  MoveL 1350 to (235.6, 160.89, 31.63) mm, rotated rx 180 ry 0 rz 180 deg; joints [-30.149, 31.04, 26.19, 47.019, 43.356, -37.963]
  Call Extruder(260.06527)
  MoveL 1351 to (235.35, 161.1, 31.63) mm, rotated rx -180 ry 0 rz 180 deg; joints [-30.182, 30.989, 26.274, 47.082, 43.354, -38.025]
  Call Extruder(260.39930)
  MoveL 1352 to (234.9, 161.43, 31.63) mm, rotated rx 180 ry 0 rz 180 deg; joints [-30.234, 30.885, 26.445, 47.194, 43.341, -38.14]
  MoveL 1353 to (234.9, 161.43, 31.63) mm, rotated rx 180 ry 0 rz 180 deg; joints [-30.234, 30.885, 26.445, 47.194, 43.341, -38.14]
  Call Extruder(260.73214)
  MoveL 1354 to (234.45, 161.76, 31.63) mm, rotated rx 180 ry 0 rz 180 deg; joints [-30.287, 30.782, 26.613, 47.306, 43.329, -38.255]
  MoveL 1355 to (234.45, 161.76, 31.63) mm, rotated rx 180 ry 0 rz 180 deg; joints [-30.287, 30.782, 26.613, 47.306, 43.329, -38.255]
  Call Extruder(260.91134)
  MoveL 1356 to (234.21, 161.94, 31.63) mm, rotated rx 180 ry 0 rz 180 deg; joints [-30.316, 30.726, 26.705, 47.366, 43.322, -38.316]
  MoveL 1357 to (234.21, 161.94, 31.63) mm, rotated rx 180 ry 0 rz 180 deg; joints [-30.316, 30.726, 26.705, 47.366, 43.322, -38.316]
  Call Extruder(261.11946)
  MoveL 1358 to (233.9, 162.11, 31.63) mm, rotated rx 180 ry 0 rz 180 deg; joints [-30.347, 30.648, 26.833, 47.441, 43.308, -38.396]
  MoveL 1359 to (233.9, 162.11, 31.63) mm, rotated rx 180 ry 0 rz 180 deg; joints [-30.347, 30.648, 26.833, 47.441, 43.308, -38.396]
  Call Extruder(261.32679)
  MoveL 1360 to (233.6, 162.29, 31.63) mm, rotated rx -180 ry 0 rz -180 deg; joints [-30.379, 30.57, 26.96, 47.515, 43.295, -38.475]
  MoveL 1361 to (233.6, 162.29, 31.63) mm, rotated rx -180 ry 0 rz -180 deg; joints [-30.379, 30.57, 26.96, 47.515, 43.295, -38.475]
  Call Extruder(261.53335)
  MoveL 1362 to (233.29, 162.46, 31.63) mm, rotated rx -180 ry 0 rz 180 deg; joints [-30.41, 30.494, 27.085, 47.589, 43.281, -38.554]
  MoveL 1363 to (233.29, 162.46, 31.63) mm, rotated rx -180 ry 0 rz 180 deg; joints [-30.41, 30.494, 27.085, 47.589, 43.281, -38.554]
  Call Extruder(261.73913)
  MoveL 1364 to (232.99, 162.64, 31.63) mm, rotated rx -180 ry 0 rz 180 deg; joints [-30.442, 30.417, 27.21, 47.663, 43.269, -38.632]
  MoveL 1365 to (232.99, 162.64, 31.63) mm, rotated rx -180 ry 0 rz 180 deg; joints [-30.442, 30.417, 27.21, 47.663, 43.269, -38.632]
  Call Extruder(261.89741)
  MoveL 1366 to (232.74, 162.74, 31.63) mm, rotated rx 180 ry 0 rz -180 deg; joints [-30.464, 30.347, 27.324, 47.724, 43.253, -38.698]
  MoveL 1367 to (232.74, 162.74, 31.63) mm, rotated rx 180 ry 0 rz -180 deg; joints [-30.464, 30.347, 27.324, 47.724, 43.253, -38.698]
  Call Extruder(262.05508)
  MoveL 1368 to (232.49, 162.85, 31.63) mm, rotated rx -180 ry 0 rz 180 deg; joints [-30.487, 30.277, 27.438, 47.784, 43.238, -38.764]
  MoveL 1369 to (232.49, 162.85, 31.63) mm, rotated rx -180 ry 0 rz 180 deg; joints [-30.487, 30.277, 27.438, 47.784, 43.238, -38.764]
  Call Extruder(262.22517)
  MoveL 1370 to (232.22, 162.97, 31.63) mm, rotated rx 180 ry 0 rz -180 deg; joints [-30.511, 30.202, 27.56, 47.849, 43.222, -38.835]
  MoveL 1371 to (232.22, 162.97, 31.63) mm, rotated rx 180 ry 0 rz -180 deg; joints [-30.511, 30.202, 27.56, 47.849, 43.222, -38.835]
  Call Extruder(262.40753)
  MoveL 1372 to (231.93, 163.09, 31.63) mm, rotated rx 180 ry 0 rz 180 deg; joints [-30.538, 30.12, 27.692, 47.918, 43.204, -38.912]
  MoveL 1373 to (231.93, 163.09, 31.63) mm, rotated rx 180 ry 0 rz 180 deg; joints [-30.538, 30.12, 27.692, 47.918, 43.204, -38.912]
  Call Extruder(262.58914)
  MoveL 1374 to (231.64, 163.21, 31.63) mm, rotated rx 180 ry 0 rz 180 deg; joints [-30.564, 30.04, 27.823, 47.988, 43.187, -38.988]
  MoveL 1375 to (231.64, 163.21, 31.63) mm, rotated rx 180 ry 0 rz 180 deg; joints [-30.564, 30.04, 27.823, 47.988, 43.187, -38.988]
  Call Extruder(262.70258)
  MoveL 1376 to (231.45, 163.27, 31.63) mm, rotated rx -180 ry 0 rz 180 deg; joints [-30.579, 29.984, 27.912, 48.032, 43.174, -39.038]
  MoveL 1377 to (231.45, 163.27, 31.63) mm, rotated rx -180 ry 0 rz 180 deg; joints [-30.579, 29.984, 27.912, 48.032, 43.174, -39.038]
  Call Extruder(262.81558)
  MoveL 1378 to (231.26, 163.33, 31.63) mm, rotated rx 180 ry 0 rz 180 deg; joints [-30.595, 29.929, 28.002, 48.077, 43.161, -39.087]
  MoveL 1379 to (231.26, 163.33, 31.63) mm, rotated rx 180 ry 0 rz 180 deg; joints [-30.595, 29.929, 28.002, 48.077, 43.161, -39.087]
  Call Extruder(262.92814)
  MoveL 1380 to (231.07, 163.39, 31.63) mm, rotated rx 180 ry 0 rz 180 deg; joints [-30.61, 29.875, 28.09, 48.121, 43.148, -39.137]
  MoveL 1381 to (231.07, 163.39, 31.63) mm, rotated rx 180 ry 0 rz 180 deg; joints [-30.61, 29.875, 28.09, 48.121, 43.148, -39.137]
  Call Extruder(263.04025)
  MoveL 1382 to (230.88, 163.45, 31.63) mm, rotated rx 180 ry 0 rz 180 deg; joints [-30.625, 29.82, 28.178, 48.165, 43.135, -39.186]
  MoveL 1383 to (230.88, 163.45, 31.63) mm, rotated rx 180 ry 0 rz 180 deg; joints [-30.625, 29.82, 28.178, 48.165, 43.135, -39.186]
  Call Extruder(263.15191)
  MoveL 1384 to (230.7, 163.51, 31.63) mm, rotated rx 180 ry 0 rz 180 deg; joints [-30.641, 29.766, 28.265, 48.209, 43.123, -39.235]
  MoveL 1385 to (230.7, 163.51, 31.63) mm, rotated rx 180 ry 0 rz 180 deg; joints [-30.641, 29.766, 28.265, 48.209, 43.123, -39.235]
  Call Extruder(263.28301)
  MoveL 1386 to (230.47, 163.58, 31.63) mm, rotated rx 180 ry 0 rz 180 deg; joints [-30.659, 29.701, 28.37, 48.261, 43.108, -39.293]
  MoveL 1387 to (230.47, 163.58, 31.63) mm, rotated rx 180 ry 0 rz 180 deg; joints [-30.659, 29.701, 28.37, 48.261, 43.108, -39.293]
  Call Extruder(263.41354)
  MoveL 1388 to (230.25, 163.65, 31.63) mm, rotated rx 180 ry 0 rz -180 deg; joints [-30.677, 29.636, 28.474, 48.313, 43.093, -39.351]
  MoveL 1389 to (230.25, 163.65, 31.63) mm, rotated rx 180 ry 0 rz -180 deg; joints [-30.677, 29.636, 28.474, 48.313, 43.093, -39.351]
  Call Extruder(263.54350)
  MoveL 1390 to (230.02, 163.72, 31.63) mm, rotated rx -180 ry 0 rz 180 deg; joints [-30.694, 29.572, 28.577, 48.364, 43.078, -39.408]
  MoveL 1391 to (230.02, 163.72, 31.63) mm, rotated rx -180 ry 0 rz 180 deg; joints [-30.694, 29.572, 28.577, 48.364, 43.078, -39.408]
  Call Extruder(263.67290)
  MoveL 1392 to (229.8, 163.78, 31.63) mm, rotated rx 180 ry 0 rz 180 deg; joints [-30.712, 29.508, 28.68, 48.415, 43.064, -39.466]
  MoveL 1393 to (229.8, 163.78, 31.63) mm, rotated rx 180 ry 0 rz 180 deg; joints [-30.712, 29.508, 28.68, 48.415, 43.064, -39.466]
  Call Extruder(263.79488)
  MoveL 1394 to (229.59, 163.84, 31.63) mm, rotated rx 180 ry 0 rz 180 deg; joints [-30.729, 29.445, 28.78, 48.464, 43.049, -39.521]
  MoveL 1395 to (229.59, 163.84, 31.63) mm, rotated rx 180 ry 0 rz 180 deg; joints [-30.729, 29.445, 28.78, 48.464, 43.049, -39.521]
  Call Extruder(263.90973)
  MoveL 1396 to (229.38, 163.88, 31.63) mm, rotated rx 180 ry 0 rz 180 deg; joints [-30.744, 29.384, 28.878, 48.511, 43.034, -39.573]
  MoveL 1397 to (229.38, 163.88, 31.63) mm, rotated rx 180 ry 0 rz 180 deg; joints [-30.744, 29.384, 28.878, 48.511, 43.034, -39.573]
  Call Extruder(264.02412)
  MoveL 1398 to (229.18, 163.93, 31.63) mm, rotated rx 180 ry 0 rz 180 deg; joints [-30.758, 29.324, 28.976, 48.557, 43.019, -39.626]
  MoveL 1399 to (229.18, 163.93, 31.63) mm, rotated rx 180 ry 0 rz 180 deg; joints [-30.758, 29.324, 28.976, 48.557, 43.019, -39.626]
  Call Extruder(264.13806)
  MoveL 1400 to (228.97, 163.97, 31.63) mm, rotated rx -180 ry 0 rz 180 deg; joints [-30.773, 29.263, 29.073, 48.603, 43.005, -39.678]
  MoveL 1401 to (228.97, 163.97, 31.63) mm, rotated rx -180 ry 0 rz 180 deg; joints [-30.773, 29.263, 29.073, 48.603, 43.005, -39.678]
  Call Extruder(264.25155)
  MoveL 1402 to (228.77, 164.02, 31.63) mm, rotated rx 180 ry 0 rz 180 deg; joints [-30.788, 29.203, 29.169, 48.648, 42.99, -39.73]
  MoveL 1403 to (228.77, 164.02, 31.63) mm, rotated rx 180 ry 0 rz 180 deg; joints [-30.788, 29.203, 29.169, 48.648, 42.99, -39.73]
  Call Extruder(264.38884)
  MoveL 1404 to (228.52, 164.07, 31.63) mm, rotated rx 180 ry 0 rz 180 deg; joints [-30.806, 29.129, 29.287, 48.704, 42.973, -39.793]
  MoveL 1405 to (228.52, 164.07, 31.63) mm, rotated rx 180 ry 0 rz 180 deg; joints [-30.806, 29.129, 29.287, 48.704, 42.973, -39.793]
  Call Extruder(264.52551)
  MoveL 1406 to (228.27, 164.12, 31.63) mm, rotated rx -180 ry 0 rz 180 deg; joints [-30.823, 29.055, 29.404, 48.759, 42.955, -39.856]
  MoveL 1407 to (228.27, 164.12, 31.63) mm, rotated rx -180 ry 0 rz 180 deg; joints [-30.823, 29.055, 29.404, 48.759, 42.955, -39.856]
  Call Extruder(264.66157)
  MoveL 1408 to (228.02, 164.17, 31.63) mm, rotated rx -180 ry 0 rz 180 deg; joints [-30.841, 28.982, 29.52, 48.814, 42.938, -39.919]
  MoveL 1409 to (228.02, 164.17, 31.63) mm, rotated rx -180 ry 0 rz 180 deg; joints [-30.841, 28.982, 29.52, 48.814, 42.938, -39.919]
  Call Extruder(264.79703)
  MoveL 1410 to (227.77, 164.22, 31.63) mm, rotated rx -180 ry 0 rz -180 deg; joints [-30.859, 28.91, 29.636, 48.869, 42.921, -39.981]
  MoveL 1411 to (227.77, 164.22, 31.63) mm, rotated rx -180 ry 0 rz -180 deg; joints [-30.859, 28.91, 29.636, 48.869, 42.921, -39.981]
  Call Extruder(264.93187)
  MoveL 1412 to (227.52, 164.27, 31.63) mm, rotated rx 180 ry 0 rz 180 deg; joints [-30.877, 28.838, 29.751, 48.923, 42.905, -40.042]
  MoveL 1413 to (227.52, 164.27, 31.63) mm, rotated rx 180 ry 0 rz 180 deg; joints [-30.877, 28.838, 29.751, 48.923, 42.905, -40.042]
  Call Extruder(265.06610)
  MoveL 1414 to (227.27, 164.32, 31.63) mm, rotated rx 180 ry 0 rz 180 deg; joints [-30.895, 28.766, 29.864, 48.978, 42.888, -40.104]
  MoveL 1415 to (227.27, 164.32, 31.63) mm, rotated rx 180 ry 0 rz 180 deg; joints [-30.895, 28.766, 29.864, 48.978, 42.888, -40.104]
  Call Extruder(265.19972)
  MoveL 1416 to (227.02, 164.36, 31.63) mm, rotated rx -180 ry 0 rz -180 deg; joints [-30.912, 28.695, 29.978, 49.032, 42.872, -40.165]
  MoveL 1417 to (227.02, 164.36, 31.63) mm, rotated rx -180 ry 0 rz -180 deg; joints [-30.912, 28.695, 29.978, 49.032, 42.872, -40.165]
  Call Extruder(265.36183)
  MoveL 1418 to (226.72, 164.41, 31.63) mm, rotated rx -180 ry 0 rz 180 deg; joints [-30.933, 28.606, 30.119, 49.097, 42.851, -40.24]
  MoveL 1419 to (226.72, 164.41, 31.63) mm, rotated rx -180 ry 0 rz 180 deg; joints [-30.933, 28.606, 30.119, 49.097, 42.851, -40.24]
  Call Extruder(265.52320)
  MoveL 1420 to (226.41, 164.46, 31.63) mm, rotated rx 180 ry 0 rz 180 deg; joints [-30.954, 28.517, 30.26, 49.163, 42.831, -40.314]
  MoveL 1421 to (226.41, 164.46, 31.63) mm, rotated rx 180 ry 0 rz 180 deg; joints [-30.954, 28.517, 30.26, 49.163, 42.831, -40.314]
  Call Extruder(265.68385)
  MoveL 1422 to (226.11, 164.51, 31.63) mm, rotated rx 180 ry 0 rz 180 deg; joints [-30.975, 28.429, 30.399, 49.228, 42.811, -40.388]
  MoveL 1423 to (226.11, 164.51, 31.63) mm, rotated rx 180 ry 0 rz 180 deg; joints [-30.975, 28.429, 30.399, 49.228, 42.811, -40.388]
  Call Extruder(265.84377)
  MoveL 1424 to (225.8, 164.56, 31.63) mm, rotated rx 180 ry 0 rz 180 deg; joints [-30.995, 28.341, 30.536, 49.292, 42.792, -40.462]
  MoveL 1425 to (225.8, 164.56, 31.63) mm, rotated rx 180 ry 0 rz 180 deg; joints [-30.995, 28.341, 30.536, 49.292, 42.792, -40.462]
  Call Extruder(266.00296)
  MoveL 1426 to (225.5, 164.61, 31.63) mm, rotated rx 180 ry 0 rz 180 deg; joints [-31.016, 28.255, 30.673, 49.357, 42.773, -40.535]
  MoveL 1427 to (225.5, 164.61, 31.63) mm, rotated rx 180 ry 0 rz 180 deg; joints [-31.016, 28.255, 30.673, 49.357, 42.773, -40.535]
  Call Extruder(266.16143)
  MoveL 1428 to (225.19, 164.66, 31.63) mm, rotated rx 180 ry 0 rz -180 deg; joints [-31.037, 28.168, 30.809, 49.421, 42.754, -40.607]
  MoveL 1429 to (225.19, 164.66, 31.63) mm, rotated rx 180 ry 0 rz -180 deg; joints [-31.037, 28.168, 30.809, 49.421, 42.754, -40.607]
  Call Extruder(266.36030)
  MoveL 1430 to (224.8, 164.7, 31.63) mm, rotated rx 180 ry 0 rz 180 deg; joints [-31.062, 28.057, 30.984, 49.501, 42.729, -40.699]
  MoveL 1431 to (224.8, 164.7, 31.63) mm, rotated rx 180 ry 0 rz 180 deg; joints [-31.062, 28.057, 30.984, 49.501, 42.729, -40.699]
  Call Extruder(266.55831)
  MoveL 1432 to (224.42, 164.75, 31.63) mm, rotated rx 180 ry 0 rz 180 deg; joints [-31.087, 27.946, 31.157, 49.581, 42.704, -40.79]
  MoveL 1433 to (224.42, 164.75, 31.63) mm, rotated rx 180 ry 0 rz 180 deg; joints [-31.087, 27.946, 31.157, 49.581, 42.704, -40.79]
  Call Extruder(266.75545)
  MoveL 1434 to (224.03, 164.79, 31.63) mm, rotated rx -180 ry 0 rz 180 deg; joints [-31.112, 27.837, 31.329, 49.66, 42.681, -40.88]
  MoveL 1435 to (224.03, 164.79, 31.63) mm, rotated rx -180 ry 0 rz 180 deg; joints [-31.112, 27.837, 31.329, 49.66, 42.681, -40.88]
  Call Extruder(266.95173)
  MoveL 1436 to (223.64, 164.84, 31.63) mm, rotated rx 180 ry 0 rz 180 deg; joints [-31.137, 27.728, 31.499, 49.739, 42.657, -40.97]
  MoveL 1437 to (223.64, 164.84, 31.63) mm, rotated rx 180 ry 0 rz 180 deg; joints [-31.137, 27.728, 31.499, 49.739, 42.657, -40.97]
  Call Extruder(267.19740)
  MoveL 1438 to (223.15, 164.89, 31.63) mm, rotated rx 180 ry 0 rz 180 deg; joints [-31.168, 27.591, 31.714, 49.837, 42.628, -41.082]
  MoveL 1439 to (223.15, 164.89, 31.63) mm, rotated rx 180 ry 0 rz 180 deg; joints [-31.168, 27.591, 31.714, 49.837, 42.628, -41.082]
  Call Extruder(267.49209)
  MoveL 1440 to (222.56, 164.93, 31.63) mm, rotated rx 180 ry 0 rz -180 deg; joints [-31.204, 27.424, 31.973, 49.954, 42.592, -41.216]
  MoveL 1441 to (222.56, 164.93, 31.63) mm, rotated rx 180 ry 0 rz -180 deg; joints [-31.204, 27.424, 31.973, 49.954, 42.592, -41.216]
  Call Extruder(267.78545)
  MoveL 1442 to (221.97, 164.98, 31.63) mm, rotated rx -180 ry 0 rz 180 deg; joints [-31.24, 27.26, 32.228, 50.07, 42.557, -41.349]
  MoveL 1443 to (221.97, 164.98, 31.63) mm, rotated rx -180 ry 0 rz 180 deg; joints [-31.24, 27.26, 32.228, 50.07, 42.557, -41.349]
  Call Extruder(268.21876)
  MoveL 1444 to (221.1, 165.02, 31.63) mm, rotated rx 180 ry 0 rz 180 deg; joints [-31.292, 27.015, 32.607, 50.24, 42.506, -41.544]
  MoveL 1445 to (221.1, 165.02, 31.63) mm, rotated rx 180 ry 0 rz 180 deg; joints [-31.292, 27.015, 32.607, 50.24, 42.506, -41.544]
  Call Extruder(268.79092)
  MoveL 1446 to (219.94, 165.07, 31.63) mm, rotated rx -180 ry 0 rz 180 deg; joints [-31.36, 26.694, 33.102, 50.461, 42.439, -41.797]
  MoveL 1447 to (219.94, 165.07, 31.63) mm, rotated rx -180 ry 0 rz 180 deg; joints [-31.36, 26.694, 33.102, 50.461, 42.439, -41.797]
  Call Extruder(269.21879)
  MoveL 1448 to (219.06, 165.09, 31.63) mm, rotated rx -180 ry 0 rz 180 deg; joints [-31.409, 26.454, 33.471, 50.625, 42.391, -41.985]
  Call Extruder(385.86744)
  MoveL 1449 to (-19.06, 165.09, 31.63) mm, rotated rx 180 ry 0 rz 180 deg; joints [-51.475, -7.489, 73.697, 72.194, 55.256, -60.596]
  MoveL 1450 to (-19.06, 165.09, 31.63) mm, rotated rx 180 ry 0 rz 180 deg; joints [-51.475, -7.489, 73.697, 72.194, 55.256, -60.596]
  Call Extruder(386.58306)
  MoveL 1451 to (-20.52, 165.05, 31.63) mm, rotated rx -180 ry 0 rz -180 deg; joints [-51.652, -7.624, 73.812, 72.287, 55.416, -60.634]
  MoveL 1452 to (-20.52, 165.05, 31.63) mm, rotated rx -180 ry 0 rz -180 deg; joints [-51.652, -7.624, 73.812, 72.287, 55.416, -60.634]
  Call Extruder(387.15780)
  MoveL 1453 to (-21.68, 165, 31.63) mm, rotated rx 180 ry 0 rz 180 deg; joints [-51.793, -7.733, 73.905, 72.36, 55.543, -60.663]
  MoveL 1454 to (-21.68, 165, 31.63) mm, rotated rx 180 ry 0 rz 180 deg; joints [-51.793, -7.733, 73.905, 72.36, 55.543, -60.663]
  Call Extruder(387.45117)
  MoveL 1455 to (-22.27, 164.95, 31.63) mm, rotated rx -180 ry 0 rz 180 deg; joints [-51.862, -7.791, 73.955, 72.395, 55.606, -60.676]
  MoveL 1456 to (-22.27, 164.95, 31.63) mm, rotated rx -180 ry 0 rz 180 deg; joints [-51.862, -7.791, 73.955, 72.395, 55.606, -60.676]
  Call Extruder(387.74586)
  MoveL 1457 to (-22.86, 164.91, 31.63) mm, rotated rx 180 ry 0 rz 180 deg; joints [-51.931, -7.849, 74.004, 72.431, 55.669, -60.689]
  MoveL 1458 to (-22.86, 164.91, 31.63) mm, rotated rx 180 ry 0 rz 180 deg; joints [-51.931, -7.849, 74.004, 72.431, 55.669, -60.689]
  Call Extruder(388.04189)
  MoveL 1459 to (-23.45, 164.86, 31.63) mm, rotated rx 180 ry 0 rz -180 deg; joints [-52.001, -7.906, 74.053, 72.466, 55.732, -60.703]
  MoveL 1460 to (-23.45, 164.86, 31.63) mm, rotated rx 180 ry 0 rz -180 deg; joints [-52.001, -7.906, 74.053, 72.466, 55.732, -60.703]
  Call Extruder(388.23816)
  MoveL 1461 to (-23.83, 164.82, 31.63) mm, rotated rx -180 ry 0 rz -180 deg; joints [-52.045, -7.945, 74.086, 72.489, 55.772, -60.71]
  MoveL 1462 to (-23.83, 164.82, 31.63) mm, rotated rx -180 ry 0 rz -180 deg; joints [-52.045, -7.945, 74.086, 72.489, 55.772, -60.71]
  Call Extruder(388.43530)
  MoveL 1463 to (-24.22, 164.77, 31.63) mm, rotated rx 180 ry 0 rz 180 deg; joints [-52.089, -7.985, 74.119, 72.511, 55.813, -60.718]
  MoveL 1464 to (-24.22, 164.77, 31.63) mm, rotated rx 180 ry 0 rz 180 deg; joints [-52.089, -7.985, 74.119, 72.511, 55.813, -60.718]
  Call Extruder(388.63331)
  MoveL 1465 to (-24.61, 164.73, 31.63) mm, rotated rx 180 ry 0 rz 180 deg; joints [-52.134, -8.024, 74.153, 72.533, 55.853, -60.726]
  MoveL 1466 to (-24.61, 164.73, 31.63) mm, rotated rx 180 ry 0 rz 180 deg; joints [-52.134, -8.024, 74.153, 72.533, 55.853, -60.726]
  Call Extruder(388.83219)
  MoveL 1467 to (-25, 164.68, 31.63) mm, rotated rx 180 ry 0 rz -180 deg; joints [-52.178, -8.064, 74.186, 72.556, 55.894, -60.734]
  MoveL 1468 to (-25, 164.68, 31.63) mm, rotated rx 180 ry 0 rz -180 deg; joints [-52.178, -8.064, 74.186, 72.556, 55.894, -60.734]
  Call Extruder(389.01127)
  MoveL 1469 to (-25.34, 164.63, 31.63) mm, rotated rx 180 ry 0 rz 180 deg; joints [-52.218, -8.099, 74.217, 72.575, 55.93, -60.741]
  MoveL 1470 to (-25.34, 164.63, 31.63) mm, rotated rx 180 ry 0 rz 180 deg; joints [-52.218, -8.099, 74.217, 72.575, 55.93, -60.741]
  Call Extruder(389.17046)
  MoveL 1471 to (-25.65, 164.58, 31.63) mm, rotated rx 180 ry 0 rz 180 deg; joints [-52.251, -8.132, 74.244, 72.592, 55.961, -60.746]
  MoveL 1472 to (-25.65, 164.58, 31.63) mm, rotated rx 180 ry 0 rz 180 deg; joints [-52.251, -8.132, 74.244, 72.592, 55.961, -60.746]
  Call Extruder(389.33039)
  MoveL 1473 to (-25.96, 164.54, 31.63) mm, rotated rx 180 ry 0 rz 180 deg; joints [-52.286, -8.164, 74.271, 72.609, 55.992, -60.752]
  MoveL 1474 to (-25.96, 164.54, 31.63) mm, rotated rx 180 ry 0 rz 180 deg; joints [-52.286, -8.164, 74.271, 72.609, 55.992, -60.752]
  Call Extruder(389.49104)
  MoveL 1475 to (-26.26, 164.49, 31.63) mm, rotated rx -180 ry 0 rz -180 deg; joints [-52.32, -8.197, 74.299, 72.626, 56.023, -60.757]
  MoveL 1476 to (-26.26, 164.49, 31.63) mm, rotated rx -180 ry 0 rz -180 deg; joints [-52.32, -8.197, 74.299, 72.626, 56.023, -60.757]
  Call Extruder(389.65242)
  MoveL 1477 to (-26.57, 164.44, 31.63) mm, rotated rx 180 ry 0 rz 180 deg; joints [-52.354, -8.229, 74.326, 72.643, 56.055, -60.762]
  MoveL 1478 to (-26.57, 164.44, 31.63) mm, rotated rx 180 ry 0 rz 180 deg; joints [-52.354, -8.229, 74.326, 72.643, 56.055, -60.762]
  Call Extruder(389.81452)
  MoveL 1479 to (-26.87, 164.39, 31.63) mm, rotated rx 180 ry 0 rz 180 deg; joints [-52.388, -8.261, 74.353, 72.66, 56.086, -60.768]
  MoveL 1480 to (-26.87, 164.39, 31.63) mm, rotated rx 180 ry 0 rz 180 deg; joints [-52.388, -8.261, 74.353, 72.66, 56.086, -60.768]
  Call Extruder(389.96273)
  MoveL 1481 to (-27.15, 164.34, 31.63) mm, rotated rx 180 ry 0 rz 180 deg; joints [-52.418, -8.291, 74.378, 72.675, 56.114, -60.772]
  MoveL 1482 to (-27.15, 164.34, 31.63) mm, rotated rx 180 ry 0 rz 180 deg; joints [-52.418, -8.291, 74.378, 72.675, 56.114, -60.772]
  Call Extruder(390.09696)
  MoveL 1483 to (-27.4, 164.29, 31.63) mm, rotated rx -180 ry 0 rz 180 deg; joints [-52.445, -8.318, 74.401, 72.688, 56.139, -60.776]
  MoveL 1484 to (-27.4, 164.29, 31.63) mm, rotated rx -180 ry 0 rz 180 deg; joints [-52.445, -8.318, 74.401, 72.688, 56.139, -60.776]
  Call Extruder(390.23180)
  MoveL 1485 to (-27.65, 164.24, 31.63) mm, rotated rx -180 ry 0 rz 180 deg; joints [-52.472, -8.346, 74.424, 72.701, 56.164, -60.78]
  MoveL 1486 to (-27.65, 164.24, 31.63) mm, rotated rx -180 ry 0 rz 180 deg; joints [-52.472, -8.346, 74.424, 72.701, 56.164, -60.78]
  Call Extruder(390.36725)
  MoveL 1487 to (-27.9, 164.19, 31.63) mm, rotated rx -180 ry 0 rz 180 deg; joints [-52.499, -8.373, 74.447, 72.714, 56.189, -60.784]
  MoveL 1488 to (-27.9, 164.19, 31.63) mm, rotated rx -180 ry 0 rz 180 deg; joints [-52.499, -8.373, 74.447, 72.714, 56.189, -60.784]
  Call Extruder(390.50331)
  MoveL 1489 to (-28.15, 164.14, 31.63) mm, rotated rx -180 ry 0 rz 180 deg; joints [-52.526, -8.4, 74.47, 72.727, 56.213, -60.788]
  MoveL 1490 to (-28.15, 164.14, 31.63) mm, rotated rx -180 ry 0 rz 180 deg; joints [-52.526, -8.4, 74.47, 72.727, 56.213, -60.788]
  Call Extruder(390.63999)
  MoveL 1491 to (-28.4, 164.09, 31.63) mm, rotated rx 180 ry 0 rz -180 deg; joints [-52.553, -8.428, 74.493, 72.74, 56.238, -60.792]
  MoveL 1492 to (-28.4, 164.09, 31.63) mm, rotated rx 180 ry 0 rz -180 deg; joints [-52.553, -8.428, 74.493, 72.74, 56.238, -60.792]
  Call Extruder(390.77727)
  MoveL 1493 to (-28.64, 164.04, 31.63) mm, rotated rx 180 ry 0 rz 180 deg; joints [-52.58, -8.455, 74.516, 72.753, 56.263, -60.795]
  MoveL 1494 to (-28.64, 164.04, 31.63) mm, rotated rx 180 ry 0 rz 180 deg; joints [-52.58, -8.455, 74.516, 72.753, 56.263, -60.795]
  Call Extruder(390.90294)
  MoveL 1495 to (-28.87, 164, 31.63) mm, rotated rx 180 ry 0 rz 180 deg; joints [-52.605, -8.48, 74.537, 72.765, 56.286, -60.799]
  MoveL 1496 to (-28.87, 164, 31.63) mm, rotated rx 180 ry 0 rz 180 deg; joints [-52.605, -8.48, 74.537, 72.765, 56.286, -60.799]
  Call Extruder(391.01688)
  MoveL 1497 to (-29.08, 163.95, 31.63) mm, rotated rx 180 ry 0 rz 180 deg; joints [-52.627, -8.503, 74.556, 72.775, 56.306, -60.802]
  MoveL 1498 to (-29.08, 163.95, 31.63) mm, rotated rx 180 ry 0 rz 180 deg; joints [-52.627, -8.503, 74.556, 72.775, 56.306, -60.802]
  Call Extruder(391.13127)
  MoveL 1499 to (-29.28, 163.91, 31.63) mm, rotated rx 180 ry 0 rz 180 deg; joints [-52.649, -8.525, 74.575, 72.786, 56.326, -60.804]
  MoveL 1500 to (-29.28, 163.91, 31.63) mm, rotated rx 180 ry 0 rz 180 deg; joints [-52.649, -8.525, 74.575, 72.786, 56.326, -60.804]
  Call Extruder(391.24612)
  MoveL 1501 to (-29.48, 163.86, 31.63) mm, rotated rx 180 ry 0 rz -180 deg; joints [-52.67, -8.548, 74.594, 72.796, 56.346, -60.807]
  MoveL 1502 to (-29.48, 163.86, 31.63) mm, rotated rx 180 ry 0 rz -180 deg; joints [-52.67, -8.548, 74.594, 72.796, 56.346, -60.807]
  Call Extruder(391.36141)
  MoveL 1503 to (-29.69, 163.82, 31.63) mm, rotated rx 180 ry 0 rz 180 deg; joints [-52.692, -8.571, 74.613, 72.807, 56.366, -60.81]
  MoveL 1504 to (-29.69, 163.82, 31.63) mm, rotated rx 180 ry 0 rz 180 deg; joints [-52.692, -8.571, 74.613, 72.807, 56.366, -60.81]
  Call Extruder(391.49081)
  MoveL 1505 to (-29.91, 163.75, 31.63) mm, rotated rx 180 ry 0 rz 180 deg; joints [-52.714, -8.598, 74.636, 72.817, 56.387, -60.812]
  MoveL 1506 to (-29.91, 163.75, 31.63) mm, rotated rx 180 ry 0 rz 180 deg; joints [-52.714, -8.598, 74.636, 72.817, 56.387, -60.812]
  Call Extruder(391.62077)
  MoveL 1507 to (-30.14, 163.68, 31.63) mm, rotated rx -180 ry 0 rz 180 deg; joints [-52.737, -8.625, 74.658, 72.827, 56.408, -60.814]
  MoveL 1508 to (-30.14, 163.68, 31.63) mm, rotated rx -180 ry 0 rz 180 deg; joints [-52.737, -8.625, 74.658, 72.827, 56.408, -60.814]
  Call Extruder(391.75130)
  MoveL 1509 to (-30.36, 163.62, 31.63) mm, rotated rx -180 ry 0 rz 180 deg; joints [-52.759, -8.652, 74.681, 72.837, 56.429, -60.816]
  MoveL 1510 to (-30.36, 163.62, 31.63) mm, rotated rx -180 ry 0 rz 180 deg; joints [-52.759, -8.652, 74.681, 72.837, 56.429, -60.816]
  Call Extruder(391.88239)
  MoveL 1511 to (-30.58, 163.55, 31.63) mm, rotated rx 180 ry 0 rz 180 deg; joints [-52.781, -8.679, 74.704, 72.847, 56.449, -60.819]
  MoveL 1512 to (-30.58, 163.55, 31.63) mm, rotated rx 180 ry 0 rz 180 deg; joints [-52.781, -8.679, 74.704, 72.847, 56.449, -60.819]
  Call Extruder(392.00403)
  MoveL 1513 to (-30.79, 163.48, 31.63) mm, rotated rx 180 ry 0 rz 180 deg; joints [-52.801, -8.704, 74.725, 72.857, 56.468, -60.82]
  MoveL 1514 to (-30.79, 163.48, 31.63) mm, rotated rx 180 ry 0 rz 180 deg; joints [-52.801, -8.704, 74.725, 72.857, 56.468, -60.82]
  Call Extruder(392.11615)
  MoveL 1515 to (-30.98, 163.42, 31.63) mm, rotated rx 180 ry 0 rz 180 deg; joints [-52.82, -8.727, 74.744, 72.865, 56.485, -60.822]
  MoveL 1516 to (-30.98, 163.42, 31.63) mm, rotated rx 180 ry 0 rz 180 deg; joints [-52.82, -8.727, 74.744, 72.865, 56.485, -60.822]
  Call Extruder(392.22871)
  MoveL 1517 to (-31.17, 163.36, 31.63) mm, rotated rx 180 ry 0 rz 180 deg; joints [-52.838, -8.75, 74.763, 72.873, 56.503, -60.823]
  MoveL 1518 to (-31.17, 163.36, 31.63) mm, rotated rx 180 ry 0 rz 180 deg; joints [-52.838, -8.75, 74.763, 72.873, 56.503, -60.823]
  Call Extruder(392.34171)
  MoveL 1519 to (-31.35, 163.3, 31.63) mm, rotated rx 180 ry 0 rz 180 deg; joints [-52.856, -8.774, 74.782, 72.882, 56.52, -60.825]
  MoveL 1520 to (-31.35, 163.3, 31.63) mm, rotated rx 180 ry 0 rz 180 deg; joints [-52.856, -8.774, 74.782, 72.882, 56.52, -60.825]
  Call Extruder(392.45516)
  MoveL 1521 to (-31.54, 163.24, 31.63) mm, rotated rx 180 ry 0 rz 180 deg; joints [-52.875, -8.797, 74.802, 72.89, 56.537, -60.826]
  MoveL 1522 to (-31.54, 163.24, 31.63) mm, rotated rx 180 ry 0 rz 180 deg; joints [-52.875, -8.797, 74.802, 72.89, 56.537, -60.826]
  Call Extruder(392.60280)
  MoveL 1523 to (-31.78, 163.15, 31.63) mm, rotated rx -180 ry 0 rz -180 deg; joints [-52.897, -8.828, 74.828, 72.9, 56.558, -60.828]
  MoveL 1524 to (-31.78, 163.15, 31.63) mm, rotated rx -180 ry 0 rz -180 deg; joints [-52.897, -8.828, 74.828, 72.9, 56.558, -60.828]
  Call Extruder(392.78516)
  MoveL 1525 to (-32.08, 163.02, 31.63) mm, rotated rx -180 ry 0 rz 180 deg; joints [-52.923, -8.867, 74.86, 72.911, 56.582, -60.828]
  MoveL 1526 to (-32.08, 163.02, 31.63) mm, rotated rx -180 ry 0 rz 180 deg; joints [-52.923, -8.867, 74.86, 72.911, 56.582, -60.828]
  Call Extruder(392.96827)
  MoveL 1527 to (-32.37, 162.9, 31.63) mm, rotated rx 180 ry 0 rz 180 deg; joints [-52.949, -8.905, 74.892, 72.922, 56.607, -60.829]
  MoveL 1528 to (-32.37, 162.9, 31.63) mm, rotated rx 180 ry 0 rz 180 deg; joints [-52.949, -8.905, 74.892, 72.922, 56.607, -60.829]
  Call Extruder(393.12594)
  MoveL 1529 to (-32.62, 162.8, 31.63) mm, rotated rx -180 ry 0 rz 180 deg; joints [-52.971, -8.939, 74.92, 72.931, 56.628, -60.83]
  MoveL 1530 to (-32.62, 162.8, 31.63) mm, rotated rx -180 ry 0 rz 180 deg; joints [-52.971, -8.939, 74.92, 72.931, 56.628, -60.83]
  Call Extruder(393.28422)
  MoveL 1531 to (-32.87, 162.69, 31.63) mm, rotated rx -180 ry 0 rz 180 deg; joints [-52.993, -8.972, 74.948, 72.94, 56.649, -60.83]
  MoveL 1532 to (-32.87, 162.69, 31.63) mm, rotated rx -180 ry 0 rz 180 deg; joints [-52.993, -8.972, 74.948, 72.94, 56.649, -60.83]
  Call Extruder(393.46623)
  MoveL 1533 to (-33.14, 162.55, 31.63) mm, rotated rx -180 ry 0 rz 180 deg; joints [-53.015, -9.012, 74.981, 72.949, 56.67, -60.83]
  MoveL 1534 to (-33.14, 162.55, 31.63) mm, rotated rx -180 ry 0 rz 180 deg; joints [-53.015, -9.012, 74.981, 72.949, 56.67, -60.83]
  Call Extruder(393.67279)
  MoveL 1535 to (-33.45, 162.37, 31.63) mm, rotated rx 180 ry 0 rz 180 deg; joints [-53.038, -9.058, 75.019, 72.957, 56.692, -60.828]
  MoveL 1536 to (-33.45, 162.37, 31.63) mm, rotated rx 180 ry 0 rz 180 deg; joints [-53.038, -9.058, 75.019, 72.957, 56.692, -60.828]
  Call Extruder(393.88012)
  MoveL 1537 to (-33.75, 162.2, 31.63) mm, rotated rx 180 ry 0 rz -180 deg; joints [-53.06, -9.104, 75.057, 72.965, 56.714, -60.826]
  MoveL 1538 to (-33.75, 162.2, 31.63) mm, rotated rx 180 ry 0 rz -180 deg; joints [-53.06, -9.104, 75.057, 72.965, 56.714, -60.826]
  Call Extruder(394.08824)
  MoveL 1539 to (-34.05, 162.02, 31.63) mm, rotated rx 180 ry 0 rz -180 deg; joints [-53.083, -9.15, 75.095, 72.973, 56.736, -60.824]
  MoveL 1540 to (-34.05, 162.02, 31.63) mm, rotated rx 180 ry 0 rz -180 deg; joints [-53.083, -9.15, 75.095, 72.973, 56.736, -60.824]
  Call Extruder(394.20594)
  MoveL 1541 to (-34.23, 161.92, 31.63) mm, rotated rx 180 ry 0 rz 180 deg; joints [-53.095, -9.176, 75.116, 72.978, 56.748, -60.823]
  MoveL 1542 to (-34.23, 161.92, 31.63) mm, rotated rx 180 ry 0 rz 180 deg; joints [-53.095, -9.176, 75.116, 72.978, 56.748, -60.823]
  Call Extruder(394.53878)
  MoveL 1543 to (-34.68, 161.59, 31.63) mm, rotated rx -180 ry 0 rz 180 deg; joints [-53.122, -9.252, 75.178, 72.985, 56.776, -60.816]
  MoveL 1544 to (-34.68, 161.59, 31.63) mm, rotated rx -180 ry 0 rz 180 deg; joints [-53.122, -9.252, 75.178, 72.985, 56.776, -60.816]
  Call Extruder(394.87281)
  MoveL 1545 to (-35.13, 161.27, 31.63) mm, rotated rx 180 ry 0 rz 180 deg; joints [-53.149, -9.327, 75.241, 72.992, 56.803, -60.81]
  MoveL 1546 to (-35.13, 161.27, 31.63) mm, rotated rx 180 ry 0 rz 180 deg; joints [-53.149, -9.327, 75.241, 72.992, 56.803, -60.81]
  Call Extruder(395.04040)
  MoveL 1547 to (-35.35, 161.1, 31.63) mm, rotated rx 180 ry 0 rz 180 deg; joints [-53.163, -9.365, 75.272, 72.996, 56.817, -60.806]
  Call Extruder(395.86969)
  MoveL 1548 to (-36.39, 160.19, 31.63) mm, rotated rx 180 ry 0 rz 180 deg; joints [-53.209, -9.556, 75.429, 73.002, 56.868, -60.782]
  Call Extruder(396.50077)
  MoveL 1549 to (-37.09, 159.41, 31.63) mm, rotated rx 180 ry 0 rz 180 deg; joints [-53.224, -9.704, 75.549, 72.993, 56.889, -60.755]
  MoveL 1550 to (-37.09, 159.41, 31.63) mm, rotated rx 180 ry 0 rz 180 deg; joints [-53.224, -9.704, 75.549, 72.993, 56.889, -60.755]
  Call Extruder(396.69836)
  MoveL 1551 to (-37.3, 159.15, 31.63) mm, rotated rx 180 ry 0 rz -180 deg; joints [-53.227, -9.751, 75.587, 72.99, 56.894, -60.747]
  Call Extruder(397.03238)
  MoveL 1552 to (-37.63, 158.7, 31.63) mm, rotated rx 180 ry 0 rz -180 deg; joints [-53.226, -9.83, 75.651, 72.98, 56.897, -60.729]
  MoveL 1553 to (-37.63, 158.7, 31.63) mm, rotated rx 180 ry 0 rz -180 deg; joints [-53.226, -9.83, 75.651, 72.98, 56.897, -60.729]
  Call Extruder(397.26956)
  MoveL 1554 to (-37.86, 158.38, 31.63) mm, rotated rx 180 ry 0 rz 180 deg; joints [-53.225, -9.886, 75.697, 72.973, 56.9, -60.717]
  Set speed (130.0 mm/s)
  MoveL 1555 to (-39.51, 155.42, 31.63) mm, rotated rx 180 ry 0 rz 180 deg; joints [-53.149, -10.357, 76.077, 72.871, 56.86, -60.589]
  MoveL 1556 to (-39.5, 155.42, 41.04) mm, rotated rx -180 ry 0 rz 180 deg; joints [-53.149, -11.319, 78.45, 73.761, 56.454, -62.206]
  Call Extruder(395.26956)
  Set speed (40.0 mm/s)
  MoveL 1557 to (-39.5, 155.42, 41.04) mm, rotated rx -180 ry 0 rz 180 deg; joints [-53.149, -11.319, 78.45, 73.761, 56.454, -62.206]
  Call Extruder(0.00000)
  Set speed (130.0 mm/s)
  MoveL 1558 to (-39.41, 155.44, 41.03) mm, rotated rx -180 ry 0 rz 180 deg; joints [-53.137, -11.309, 78.442, 73.755, 56.444, -62.205]
  Call Extruder(2.00000)
  Set speed (40.0 mm/s)
  MoveL 1559 to (-39.41, 155.44, 41.03) mm, rotated rx -180 ry 0 rz 180 deg; joints [-53.137, -11.309, 78.442, 73.755, 56.444, -62.205]
  Set speed (30.0 mm/s)
  MoveL 1560 to (-39.41, 155.44, 41.03) mm, rotated rx -180 ry 0 rz 180 deg; joints [-53.137, -11.309, 78.442, 73.755, 56.444, -62.205]
  Call Extruder(2.05684)
  MoveL 1561 to (-39.44, 155.34, 41.04) mm, rotated rx 180 ry 0 rz 180 deg; joints [-53.131, -11.322, 78.453, 73.75, 56.439, -62.2]
  MoveL 1562 to (-39.44, 155.34, 41.04) mm, rotated rx 180 ry 0 rz 180 deg; joints [-53.131, -11.322, 78.453, 73.75, 56.439, -62.2]
  Call Extruder(2.17007)
  MoveL 1563 to (-39.5, 155.15, 41.04) mm, rotated rx -180 ry 0 rz 180 deg; joints [-53.121, -11.349, 78.473, 73.741, 56.432, -62.19]
  MoveL 1564 to (-39.5, 155.15, 41.04) mm, rotated rx -180 ry 0 rz 180 deg; joints [-53.121, -11.349, 78.473, 73.741, 56.432, -62.19]
  Call Extruder(2.28286)
  MoveL 1565 to (-39.56, 154.97, 41.04) mm, rotated rx 180 ry 0 rz 180 deg; joints [-53.11, -11.375, 78.494, 73.731, 56.424, -62.181]
  MoveL 1566 to (-39.56, 154.97, 41.04) mm, rotated rx 180 ry 0 rz 180 deg; joints [-53.11, -11.375, 78.494, 73.731, 56.424, -62.181]
  Call Extruder(2.39521)
  MoveL 1567 to (-39.62, 154.78, 41.04) mm, rotated rx 180 ry 0 rz 180 deg; joints [-53.099, -11.401, 78.515, 73.722, 56.416, -62.171]
  MoveL 1568 to (-39.62, 154.78, 41.04) mm, rotated rx 180 ry 0 rz 180 deg; joints [-53.099, -11.401, 78.515, 73.722, 56.416, -62.171]
  Call Extruder(2.50711)
  MoveL 1569 to (-39.68, 154.59, 41.03) mm, rotated rx -180 ry 0 rz 180 deg; joints [-53.088, -11.427, 78.535, 73.712, 56.408, -62.161]
  MoveL 1570 to (-39.68, 154.59, 41.03) mm, rotated rx -180 ry 0 rz 180 deg; joints [-53.088, -11.427, 78.535, 73.712, 56.408, -62.161]
  Call Extruder(2.62851)
  MoveL 1571 to (-39.75, 154.38, 41.04) mm, rotated rx 180 ry 0 rz 180 deg; joints [-53.076, -11.456, 78.558, 73.701, 56.399, -62.15]
  MoveL 1572 to (-39.75, 154.38, 41.04) mm, rotated rx 180 ry 0 rz 180 deg; joints [-53.076, -11.456, 78.558, 73.701, 56.399, -62.15]
  Call Extruder(2.75930)
  MoveL 1573 to (-39.81, 154.16, 41.04) mm, rotated rx 180 ry 0 rz 180 deg; joints [-53.063, -11.487, 78.582, 73.69, 56.389, -62.138]
  MoveL 1574 to (-39.81, 154.16, 41.04) mm, rotated rx 180 ry 0 rz 180 deg; joints [-53.063, -11.487, 78.582, 73.69, 56.389, -62.138]
  Call Extruder(2.88953)
  MoveL 1575 to (-39.88, 153.94, 41.04) mm, rotated rx -180 ry 0 rz -180 deg; joints [-53.049, -11.517, 78.606, 73.678, 56.378, -62.127]
  MoveL 1576 to (-39.88, 153.94, 41.04) mm, rotated rx -180 ry 0 rz -180 deg; joints [-53.049, -11.517, 78.606, 73.678, 56.378, -62.127]
  Call Extruder(3.01920)
  MoveL 1577 to (-39.95, 153.71, 41.04) mm, rotated rx 180 ry 0 rz -180 deg; joints [-53.036, -11.548, 78.63, 73.666, 56.368, -62.115]
  MoveL 1578 to (-39.95, 153.71, 41.04) mm, rotated rx 180 ry 0 rz -180 deg; joints [-53.036, -11.548, 78.63, 73.666, 56.368, -62.115]
  Call Extruder(3.14830)
  MoveL 1579 to (-40.02, 153.49, 41.04) mm, rotated rx 180 ry 0 rz 180 deg; joints [-53.022, -11.579, 78.654, 73.654, 56.358, -62.103]
  MoveL 1580 to (-40.02, 153.49, 41.04) mm, rotated rx 180 ry 0 rz 180 deg; joints [-53.022, -11.579, 78.654, 73.654, 56.358, -62.103]
  Call Extruder(3.26338)
  MoveL 1581 to (-40.06, 153.28, 41.04) mm, rotated rx 180 ry 0 rz -180 deg; joints [-53.007, -11.605, 78.675, 73.642, 56.347, -62.092]
  MoveL 1582 to (-40.06, 153.28, 41.04) mm, rotated rx 180 ry 0 rz -180 deg; joints [-53.007, -11.605, 78.675, 73.642, 56.347, -62.092]
  Call Extruder(3.37802)
  MoveL 1583 to (-40.11, 153.08, 41.03) mm, rotated rx 180 ry 0 rz 180 deg; joints [-52.993, -11.632, 78.696, 73.63, 56.335, -62.08]
  MoveL 1584 to (-40.11, 153.08, 41.03) mm, rotated rx 180 ry 0 rz 180 deg; joints [-52.993, -11.632, 78.696, 73.63, 56.335, -62.08]
  Call Extruder(3.49220)
  MoveL 1585 to (-40.15, 152.88, 41.04) mm, rotated rx 180 ry 0 rz 180 deg; joints [-52.978, -11.658, 78.716, 73.618, 56.324, -62.069]
  MoveL 1586 to (-40.15, 152.88, 41.04) mm, rotated rx 180 ry 0 rz 180 deg; joints [-52.978, -11.658, 78.716, 73.618, 56.324, -62.069]
  Call Extruder(3.60593)
  MoveL 1587 to (-40.2, 152.67, 41.04) mm, rotated rx 180 ry 0 rz 180 deg; joints [-52.963, -11.685, 78.737, 73.606, 56.313, -62.058]
  MoveL 1588 to (-40.2, 152.67, 41.04) mm, rotated rx 180 ry 0 rz 180 deg; joints [-52.963, -11.685, 78.737, 73.606, 56.313, -62.058]
  Call Extruder(3.73136)
  MoveL 1589 to (-40.24, 152.45, 41.04) mm, rotated rx -180 ry 0 rz 180 deg; joints [-52.946, -11.714, 78.76, 73.593, 56.3, -62.045]
  MoveL 1590 to (-40.24, 152.45, 41.04) mm, rotated rx -180 ry 0 rz 180 deg; joints [-52.946, -11.714, 78.76, 73.593, 56.3, -62.045]
  Call Extruder(3.86834)
  MoveL 1591 to (-40.29, 152.2, 41.04) mm, rotated rx 180 ry 0 rz 180 deg; joints [-52.928, -11.746, 78.785, 73.578, 56.285, -62.031]
  MoveL 1592 to (-40.29, 152.2, 41.04) mm, rotated rx 180 ry 0 rz 180 deg; joints [-52.928, -11.746, 78.785, 73.578, 56.285, -62.031]
  Call Extruder(4.00470)
  MoveL 1593 to (-40.34, 151.95, 41.04) mm, rotated rx -180 ry 0 rz 180 deg; joints [-52.909, -11.778, 78.81, 73.562, 56.27, -62.017]
  MoveL 1594 to (-40.34, 151.95, 41.04) mm, rotated rx -180 ry 0 rz 180 deg; joints [-52.909, -11.778, 78.81, 73.562, 56.27, -62.017]
  Call Extruder(4.14046)
  MoveL 1595 to (-40.39, 151.7, 41.04) mm, rotated rx 180 ry 0 rz 180 deg; joints [-52.89, -11.81, 78.835, 73.547, 56.256, -62.003]
  MoveL 1596 to (-40.39, 151.7, 41.04) mm, rotated rx 180 ry 0 rz 180 deg; joints [-52.89, -11.81, 78.835, 73.547, 56.256, -62.003]
  Call Extruder(4.27560)
  MoveL 1597 to (-40.44, 151.45, 41.03) mm, rotated rx -180 ry 0 rz 180 deg; joints [-52.871, -11.842, 78.859, 73.532, 56.241, -61.989]
  MoveL 1598 to (-40.44, 151.45, 41.03) mm, rotated rx -180 ry 0 rz 180 deg; joints [-52.871, -11.842, 78.859, 73.532, 56.241, -61.989]
  Call Extruder(4.41014)
  MoveL 1599 to (-40.49, 151.2, 41.03) mm, rotated rx 180 ry 0 rz 180 deg; joints [-52.853, -11.874, 78.884, 73.517, 56.227, -61.975]
  MoveL 1600 to (-40.49, 151.2, 41.03) mm, rotated rx 180 ry 0 rz 180 deg; joints [-52.853, -11.874, 78.884, 73.517, 56.227, -61.975]
  Call Extruder(4.54406)
  MoveL 1601 to (-40.54, 150.95, 41.04) mm, rotated rx 180 ry 0 rz 180 deg; joints [-52.834, -11.906, 78.909, 73.502, 56.212, -61.961]
  MoveL 1602 to (-40.54, 150.95, 41.04) mm, rotated rx 180 ry 0 rz 180 deg; joints [-52.834, -11.906, 78.909, 73.502, 56.212, -61.961]
  Call Extruder(4.69192)
  MoveL 1603 to (-40.59, 150.67, 41.04) mm, rotated rx 180 ry 0 rz 180 deg; joints [-52.812, -11.94, 78.936, 73.485, 56.195, -61.945]
  MoveL 1604 to (-40.59, 150.67, 41.04) mm, rotated rx 180 ry 0 rz 180 deg; joints [-52.812, -11.94, 78.936, 73.485, 56.195, -61.945]
  Call Extruder(4.85364)
  MoveL 1605 to (-40.64, 150.37, 41.04) mm, rotated rx 180 ry 0 rz 180 deg; joints [-52.787, -11.979, 78.966, 73.465, 56.176, -61.928]
  MoveL 1606 to (-40.64, 150.37, 41.04) mm, rotated rx 180 ry 0 rz 180 deg; joints [-52.787, -11.979, 78.966, 73.465, 56.176, -61.928]
  Call Extruder(5.01464)
  MoveL 1607 to (-40.69, 150.06, 41.04) mm, rotated rx 180 ry 0 rz 180 deg; joints [-52.762, -12.017, 78.995, 73.445, 56.156, -61.91]
  MoveL 1608 to (-40.69, 150.06, 41.04) mm, rotated rx 180 ry 0 rz 180 deg; joints [-52.762, -12.017, 78.995, 73.445, 56.156, -61.91]
  Call Extruder(5.17491)
  MoveL 1609 to (-40.74, 149.76, 41.04) mm, rotated rx -180 ry 0 rz 180 deg; joints [-52.737, -12.055, 79.024, 73.426, 56.137, -61.892]
  MoveL 1610 to (-40.74, 149.76, 41.04) mm, rotated rx -180 ry 0 rz 180 deg; joints [-52.737, -12.055, 79.024, 73.426, 56.137, -61.892]
  Call Extruder(5.33445)
  MoveL 1611 to (-40.78, 149.45, 41.03) mm, rotated rx 180 ry 0 rz 180 deg; joints [-52.712, -12.092, 79.054, 73.406, 56.117, -61.874]
  MoveL 1612 to (-40.78, 149.45, 41.03) mm, rotated rx 180 ry 0 rz 180 deg; joints [-52.712, -12.092, 79.054, 73.406, 56.117, -61.874]
  Call Extruder(5.49326)
  MoveL 1613 to (-40.83, 149.14, 41.04) mm, rotated rx -180 ry 0 rz -180 deg; joints [-52.687, -12.13, 79.083, 73.386, 56.097, -61.856]
  MoveL 1614 to (-40.83, 149.14, 41.04) mm, rotated rx -180 ry 0 rz -180 deg; joints [-52.687, -12.13, 79.083, 73.386, 56.097, -61.856]
  Call Extruder(5.67193)
  MoveL 1615 to (-40.88, 148.8, 41.04) mm, rotated rx 180 ry 0 rz -180 deg; joints [-52.658, -12.173, 79.116, 73.363, 56.074, -61.836]
  MoveL 1616 to (-40.88, 148.8, 41.04) mm, rotated rx 180 ry 0 rz -180 deg; joints [-52.658, -12.173, 79.116, 73.363, 56.074, -61.836]
  Call Extruder(5.87037)
  MoveL 1617 to (-40.92, 148.41, 41.04) mm, rotated rx 180 ry 0 rz 180 deg; joints [-52.624, -12.219, 79.152, 73.337, 56.047, -61.813]
  MoveL 1618 to (-40.92, 148.41, 41.04) mm, rotated rx 180 ry 0 rz 180 deg; joints [-52.624, -12.219, 79.152, 73.337, 56.047, -61.813]
  Call Extruder(6.06794)
  MoveL 1619 to (-40.97, 148.02, 41.04) mm, rotated rx 180 ry 0 rz 180 deg; joints [-52.59, -12.266, 79.188, 73.311, 56.02, -61.79]
  MoveL 1620 to (-40.97, 148.02, 41.04) mm, rotated rx 180 ry 0 rz 180 deg; joints [-52.59, -12.266, 79.188, 73.311, 56.02, -61.79]
  Call Extruder(6.26465)
  MoveL 1621 to (-41.02, 147.63, 41.04) mm, rotated rx -180 ry 0 rz 180 deg; joints [-52.556, -12.313, 79.224, 73.284, 55.993, -61.766]
  MoveL 1622 to (-41.02, 147.63, 41.04) mm, rotated rx -180 ry 0 rz 180 deg; joints [-52.556, -12.313, 79.224, 73.284, 55.993, -61.766]
  Call Extruder(6.46049)
  MoveL 1623 to (-41.06, 147.25, 41.04) mm, rotated rx 180 ry 0 rz 180 deg; joints [-52.521, -12.359, 79.26, 73.258, 55.966, -61.743]
  MoveL 1624 to (-41.06, 147.25, 41.04) mm, rotated rx 180 ry 0 rz 180 deg; joints [-52.521, -12.359, 79.26, 73.258, 55.966, -61.743]
  Call Extruder(6.75588)
  MoveL 1625 to (-41.11, 146.66, 41.03) mm, rotated rx -180 ry 0 rz 180 deg; joints [-52.466, -12.428, 79.312, 73.216, 55.922, -61.707]
  MoveL 1626 to (-41.11, 146.66, 41.03) mm, rotated rx -180 ry 0 rz 180 deg; joints [-52.466, -12.428, 79.312, 73.216, 55.922, -61.707]
  Call Extruder(7.04995)
  MoveL 1627 to (-41.15, 146.07, 41.04) mm, rotated rx 180 ry 0 rz 180 deg; joints [-52.411, -12.497, 79.365, 73.174, 55.878, -61.67]
  MoveL 1628 to (-41.15, 146.07, 41.04) mm, rotated rx 180 ry 0 rz 180 deg; joints [-52.411, -12.497, 79.365, 73.174, 55.878, -61.67]
  Call Extruder(7.34268)
  MoveL 1629 to (-41.2, 145.48, 41.04) mm, rotated rx 180 ry 0 rz 180 deg; joints [-52.355, -12.566, 79.418, 73.131, 55.834, -61.634]
  MoveL 1630 to (-41.2, 145.48, 41.04) mm, rotated rx 180 ry 0 rz 180 deg; joints [-52.355, -12.566, 79.418, 73.131, 55.834, -61.634]
  Call Extruder(7.91614)
  MoveL 1631 to (-41.25, 144.32, 41.04) mm, rotated rx 180 ry 0 rz 180 deg; joints [-52.239, -12.697, 79.518, 73.044, 55.741, -61.56]
  MoveL 1632 to (-41.25, 144.32, 41.04) mm, rotated rx 180 ry 0 rz 180 deg; joints [-52.239, -12.697, 79.518, 73.044, 55.741, -61.56]
  Call Extruder(8.63010)
  MoveL 1633 to (-41.29, 142.86, 41.04) mm, rotated rx -180 ry 0 rz 180 deg; joints [-52.09, -12.859, 79.641, 72.933, 55.621, -61.467]
  Call Extruder(50.69492)
  MoveL 1634 to (-41.29, 57.14, 41.04) mm, rotated rx 180 ry 0 rz 180 deg; joints [-40.759, -21.186, 85.282, 63.121, 47.05, -53.355]
  Call Extruder(51.12347)
  MoveL 1635 to (-41.27, 56.26, 41.04) mm, rotated rx 180 ry 0 rz 180 deg; joints [-40.614, -21.258, 85.324, 62.979, 46.948, -53.239]
  MoveL 1636 to (-41.27, 56.26, 41.04) mm, rotated rx 180 ry 0 rz 180 deg; joints [-40.614, -21.258, 85.324, 62.979, 46.948, -53.239]
  Call Extruder(51.69692)
  MoveL 1637 to (-41.22, 55.1, 41.03) mm, rotated rx 180 ry 0 rz 180 deg; joints [-40.419, -21.351, 85.379, 62.787, 46.808, -53.083]
  MoveL 1638 to (-41.22, 55.1, 41.03) mm, rotated rx 180 ry 0 rz 180 deg; joints [-40.419, -21.351, 85.379, 62.787, 46.808, -53.083]
  Call Extruder(52.13124)
  MoveL 1639 to (-41.18, 54.23, 41.04) mm, rotated rx 180 ry 0 rz 180 deg; joints [-40.269, -21.419, 85.42, 62.64, 46.701, -52.964]
  MoveL 1640 to (-41.18, 54.23, 41.04) mm, rotated rx 180 ry 0 rz 180 deg; joints [-40.269, -21.419, 85.42, 62.64, 46.701, -52.964]
  Call Extruder(52.42530)
  MoveL 1641 to (-41.13, 53.64, 41.04) mm, rotated rx 180 ry 0 rz 180 deg; joints [-40.165, -21.463, 85.446, 62.539, 46.627, -52.882]
  MoveL 1642 to (-41.13, 53.64, 41.04) mm, rotated rx 180 ry 0 rz 180 deg; joints [-40.165, -21.463, 85.446, 62.539, 46.627, -52.882]
  Call Extruder(52.72070)
  MoveL 1643 to (-41.09, 53.05, 41.04) mm, rotated rx 180 ry 0 rz 180 deg; joints [-40.062, -21.508, 85.472, 62.437, 46.553, -52.801]
  MoveL 1644 to (-41.09, 53.05, 41.04) mm, rotated rx 180 ry 0 rz 180 deg; joints [-40.062, -21.508, 85.472, 62.437, 46.553, -52.801]
  Call Extruder(52.96694)
  MoveL 1645 to (-41.04, 52.56, 41.04) mm, rotated rx 180 ry 0 rz 180 deg; joints [-39.975, -21.543, 85.493, 62.352, 46.491, -52.733]
  MoveL 1646 to (-41.04, 52.56, 41.04) mm, rotated rx 180 ry 0 rz 180 deg; joints [-39.975, -21.543, 85.493, 62.352, 46.491, -52.733]
  Call Extruder(53.16365)
  MoveL 1647 to (-40.99, 52.17, 41.03) mm, rotated rx 180 ry 0 rz 180 deg; joints [-39.904, -21.571, 85.509, 62.284, 46.44, -52.679]
  MoveL 1648 to (-40.99, 52.17, 41.03) mm, rotated rx 180 ry 0 rz 180 deg; joints [-39.904, -21.571, 85.509, 62.284, 46.44, -52.679]
  Call Extruder(53.36122)
  MoveL 1649 to (-40.95, 51.78, 41.04) mm, rotated rx 180 ry 0 rz 180 deg; joints [-39.833, -21.598, 85.525, 62.215, 46.389, -52.624]
  MoveL 1650 to (-40.95, 51.78, 41.04) mm, rotated rx 180 ry 0 rz 180 deg; joints [-39.833, -21.598, 85.525, 62.215, 46.389, -52.624]
  Call Extruder(53.55966)
  MoveL 1651 to (-40.9, 51.4, 41.04) mm, rotated rx 180 ry 0 rz 180 deg; joints [-39.763, -21.625, 85.541, 62.146, 46.338, -52.569]
  MoveL 1652 to (-40.9, 51.4, 41.04) mm, rotated rx 180 ry 0 rz 180 deg; joints [-39.763, -21.625, 85.541, 62.146, 46.338, -52.569]
  Call Extruder(53.75897)
  MoveL 1653 to (-40.86, 51.01, 41.04) mm, rotated rx 180 ry 0 rz -180 deg; joints [-39.692, -21.653, 85.557, 62.077, 46.287, -52.514]
  MoveL 1654 to (-40.86, 51.01, 41.04) mm, rotated rx 180 ry 0 rz -180 deg; joints [-39.692, -21.653, 85.557, 62.077, 46.287, -52.514]
  Call Extruder(53.91779)
  MoveL 1655 to (-40.81, 50.7, 41.04) mm, rotated rx -180 ry 0 rz 180 deg; joints [-39.634, -21.673, 85.569, 62.021, 46.245, -52.47]
  MoveL 1656 to (-40.81, 50.7, 41.04) mm, rotated rx -180 ry 0 rz 180 deg; joints [-39.634, -21.673, 85.569, 62.021, 46.245, -52.47]
  Call Extruder(54.07733)
  MoveL 1657 to (-40.76, 50.4, 41.04) mm, rotated rx -180 ry 0 rz 180 deg; joints [-39.576, -21.693, 85.58, 61.965, 46.203, -52.426]
  MoveL 1658 to (-40.76, 50.4, 41.04) mm, rotated rx -180 ry 0 rz 180 deg; joints [-39.576, -21.693, 85.58, 61.965, 46.203, -52.426]
  Call Extruder(54.23760)
  MoveL 1659 to (-40.71, 50.09, 41.04) mm, rotated rx 180 ry 0 rz 180 deg; joints [-39.518, -21.713, 85.592, 61.909, 46.161, -52.382]
  MoveL 1660 to (-40.71, 50.09, 41.04) mm, rotated rx 180 ry 0 rz 180 deg; joints [-39.518, -21.713, 85.592, 61.909, 46.161, -52.382]
  Call Extruder(54.39860)
  MoveL 1661 to (-40.66, 49.79, 41.04) mm, rotated rx 180 ry 0 rz 180 deg; joints [-39.46, -21.733, 85.604, 61.853, 46.119, -52.338]
  MoveL 1662 to (-40.66, 49.79, 41.04) mm, rotated rx 180 ry 0 rz 180 deg; joints [-39.46, -21.733, 85.604, 61.853, 46.119, -52.338]
  Call Extruder(54.56032)
  MoveL 1663 to (-40.61, 49.48, 41.04) mm, rotated rx 180 ry 0 rz 180 deg; joints [-39.402, -21.754, 85.616, 61.797, 46.077, -52.293]
  MoveL 1664 to (-40.61, 49.48, 41.04) mm, rotated rx 180 ry 0 rz 180 deg; joints [-39.402, -21.754, 85.616, 61.797, 46.077, -52.293]
  Call Extruder(54.72278)
  MoveL 1665 to (-40.56, 49.18, 41.03) mm, rotated rx 180 ry 0 rz 180 deg; joints [-39.344, -21.773, 85.627, 61.74, 46.035, -52.249]
  MoveL 1666 to (-40.56, 49.18, 41.03) mm, rotated rx 180 ry 0 rz 180 deg; joints [-39.344, -21.773, 85.627, 61.74, 46.035, -52.249]
  Call Extruder(54.85670)
  MoveL 1667 to (-40.52, 48.93, 41.04) mm, rotated rx 180 ry 0 rz 180 deg; joints [-39.296, -21.789, 85.636, 61.693, 46, -52.212]
  MoveL 1668 to (-40.52, 48.93, 41.04) mm, rotated rx 180 ry 0 rz 180 deg; joints [-39.296, -21.789, 85.636, 61.693, 46, -52.212]
  Call Extruder(54.99124)
  MoveL 1669 to (-40.47, 48.68, 41.03) mm, rotated rx 180 ry 0 rz 180 deg; joints [-39.247, -21.804, 85.645, 61.646, 45.964, -52.176]
  MoveL 1670 to (-40.47, 48.68, 41.03) mm, rotated rx 180 ry 0 rz 180 deg; joints [-39.247, -21.804, 85.645, 61.646, 45.964, -52.176]
  Call Extruder(55.12638)
  MoveL 1671 to (-40.42, 48.43, 41.04) mm, rotated rx 180 ry 0 rz 180 deg; joints [-39.198, -21.819, 85.654, 61.599, 45.929, -52.139]
  MoveL 1672 to (-40.42, 48.43, 41.04) mm, rotated rx 180 ry 0 rz 180 deg; joints [-39.198, -21.819, 85.654, 61.599, 45.929, -52.139]
  Call Extruder(55.26214)
  MoveL 1673 to (-40.37, 48.18, 41.04) mm, rotated rx -180 ry 0 rz 180 deg; joints [-39.149, -21.835, 85.663, 61.552, 45.893, -52.102]
  MoveL 1674 to (-40.37, 48.18, 41.04) mm, rotated rx -180 ry 0 rz 180 deg; joints [-39.149, -21.835, 85.663, 61.552, 45.893, -52.102]
  Call Extruder(55.39850)
  MoveL 1675 to (-40.32, 47.93, 41.04) mm, rotated rx -180 ry 0 rz 180 deg; joints [-39.1, -21.85, 85.671, 61.505, 45.858, -52.065]
  MoveL 1676 to (-40.32, 47.93, 41.04) mm, rotated rx -180 ry 0 rz 180 deg; joints [-39.1, -21.85, 85.671, 61.505, 45.858, -52.065]
  Call Extruder(55.53548)
  MoveL 1677 to (-40.27, 47.68, 41.04) mm, rotated rx -180 ry 0 rz 180 deg; joints [-39.051, -21.865, 85.68, 61.457, 45.822, -52.028]
  MoveL 1678 to (-40.27, 47.68, 41.04) mm, rotated rx -180 ry 0 rz 180 deg; joints [-39.051, -21.865, 85.68, 61.457, 45.822, -52.028]
  Call Extruder(55.67306)
  MoveL 1679 to (-40.22, 47.43, 41.04) mm, rotated rx -180 ry 0 rz -180 deg; joints [-39.002, -21.88, 85.689, 61.41, 45.787, -51.991]
  MoveL 1680 to (-40.22, 47.43, 41.04) mm, rotated rx -180 ry 0 rz -180 deg; joints [-39.002, -21.88, 85.689, 61.41, 45.787, -51.991]
  Call Extruder(55.78679)
  MoveL 1681 to (-40.17, 47.23, 41.03) mm, rotated rx -180 ry 0 rz 180 deg; joints [-38.962, -21.892, 85.696, 61.371, 45.757, -51.96]
  MoveL 1682 to (-40.17, 47.23, 41.03) mm, rotated rx -180 ry 0 rz 180 deg; joints [-38.962, -21.892, 85.696, 61.371, 45.757, -51.96]
  Call Extruder(55.90097)
  MoveL 1683 to (-40.13, 47.02, 41.04) mm, rotated rx 180 ry 0 rz 180 deg; joints [-38.921, -21.904, 85.703, 61.331, 45.727, -51.929]
  MoveL 1684 to (-40.13, 47.02, 41.04) mm, rotated rx 180 ry 0 rz 180 deg; joints [-38.921, -21.904, 85.703, 61.331, 45.727, -51.929]
  Call Extruder(56.01561)
  MoveL 1685 to (-40.08, 46.82, 41.04) mm, rotated rx 180 ry 0 rz 180 deg; joints [-38.88, -21.916, 85.71, 61.291, 45.697, -51.899]
  MoveL 1686 to (-40.08, 46.82, 41.04) mm, rotated rx 180 ry 0 rz 180 deg; joints [-38.88, -21.916, 85.71, 61.291, 45.697, -51.899]
  Call Extruder(56.13069)
  MoveL 1687 to (-40.04, 46.61, 41.04) mm, rotated rx 180 ry 0 rz -180 deg; joints [-38.839, -21.928, 85.717, 61.252, 45.668, -51.868]
  MoveL 1688 to (-40.04, 46.61, 41.04) mm, rotated rx 180 ry 0 rz -180 deg; joints [-38.839, -21.928, 85.717, 61.252, 45.668, -51.868]
  Call Extruder(56.25293)
  MoveL 1689 to (-39.98, 46.4, 41.04) mm, rotated rx 180 ry 0 rz -180 deg; joints [-38.795, -21.94, 85.724, 61.21, 45.636, -51.835]
  MoveL 1690 to (-39.98, 46.4, 41.04) mm, rotated rx 180 ry 0 rz -180 deg; joints [-38.795, -21.94, 85.724, 61.21, 45.636, -51.835]
  Call Extruder(56.38259)
  MoveL 1691 to (-39.92, 46.18, 41.04) mm, rotated rx 180 ry 0 rz 180 deg; joints [-38.748, -21.951, 85.73, 61.165, 45.601, -51.801]
  MoveL 1692 to (-39.92, 46.18, 41.04) mm, rotated rx 180 ry 0 rz 180 deg; joints [-38.748, -21.951, 85.73, 61.165, 45.601, -51.801]
  Call Extruder(56.51282)
  MoveL 1693 to (-39.85, 45.95, 41.04) mm, rotated rx 180 ry 0 rz 180 deg; joints [-38.7, -21.962, 85.736, 61.12, 45.566, -51.766]
  MoveL 1694 to (-39.85, 45.95, 41.04) mm, rotated rx 180 ry 0 rz 180 deg; joints [-38.7, -21.962, 85.736, 61.12, 45.566, -51.766]
  Call Extruder(56.64361)
  MoveL 1695 to (-39.78, 45.73, 41.04) mm, rotated rx -180 ry 0 rz 180 deg; joints [-38.653, -21.973, 85.743, 61.074, 45.531, -51.732]
  MoveL 1696 to (-39.78, 45.73, 41.04) mm, rotated rx -180 ry 0 rz 180 deg; joints [-38.653, -21.973, 85.743, 61.074, 45.531, -51.732]
  Call Extruder(56.77497)
  MoveL 1697 to (-39.71, 45.51, 41.04) mm, rotated rx 180 ry 0 rz 180 deg; joints [-38.605, -21.984, 85.749, 61.029, 45.496, -51.697]
  MoveL 1698 to (-39.71, 45.51, 41.04) mm, rotated rx 180 ry 0 rz 180 deg; joints [-38.605, -21.984, 85.749, 61.029, 45.496, -51.697]
  Call Extruder(56.88687)
  MoveL 1699 to (-39.65, 45.32, 41.04) mm, rotated rx 180 ry 0 rz 180 deg; joints [-38.565, -21.993, 85.754, 60.991, 45.466, -51.668]
  MoveL 1700 to (-39.65, 45.32, 41.04) mm, rotated rx 180 ry 0 rz 180 deg; joints [-38.565, -21.993, 85.754, 60.991, 45.466, -51.668]
  Call Extruder(56.99922)
  MoveL 1701 to (-39.59, 45.13, 41.04) mm, rotated rx -180 ry 0 rz 180 deg; joints [-38.524, -22.002, 85.76, 60.952, 45.436, -51.638]
  MoveL 1702 to (-39.59, 45.13, 41.04) mm, rotated rx -180 ry 0 rz 180 deg; joints [-38.524, -22.002, 85.76, 60.952, 45.436, -51.638]
  Call Extruder(57.11201)
  MoveL 1703 to (-39.53, 44.94, 41.04) mm, rotated rx 180 ry 0 rz -180 deg; joints [-38.483, -22.011, 85.765, 60.913, 45.405, -51.609]
  MoveL 1704 to (-39.53, 44.94, 41.04) mm, rotated rx 180 ry 0 rz -180 deg; joints [-38.483, -22.011, 85.765, 60.913, 45.405, -51.609]
  Call Extruder(57.22525)
  MoveL 1705 to (-39.47, 44.75, 41.04) mm, rotated rx 180 ry 0 rz 180 deg; joints [-38.443, -22.02, 85.77, 60.875, 45.375, -51.579]
  MoveL 1706 to (-39.47, 44.75, 41.04) mm, rotated rx 180 ry 0 rz 180 deg; joints [-38.443, -22.02, 85.77, 60.875, 45.375, -51.579]
  Call Extruder(57.33893)
  MoveL 1707 to (-39.41, 44.56, 41.03) mm, rotated rx 180 ry 0 rz 180 deg; joints [-38.402, -22.028, 85.775, 60.836, 45.345, -51.55]
  MoveL 1708 to (-39.41, 44.56, 41.03) mm, rotated rx 180 ry 0 rz 180 deg; joints [-38.402, -22.028, 85.775, 60.836, 45.345, -51.55]
  Call Extruder(57.52088)
  MoveL 1709 to (-39.29, 44.27, 41.03) mm, rotated rx 180 ry 0 rz 180 deg; joints [-38.335, -22.039, 85.781, 60.774, 45.296, -51.503]
  MoveL 1710 to (-39.29, 44.27, 41.03) mm, rotated rx 180 ry 0 rz 180 deg; joints [-38.335, -22.039, 85.781, 60.774, 45.296, -51.503]
  Call Extruder(57.70360)
  MoveL 1711 to (-39.16, 43.98, 41.04) mm, rotated rx 180 ry 0 rz 180 deg; joints [-38.269, -22.05, 85.788, 60.711, 45.246, -51.456]
  MoveL 1712 to (-39.16, 43.98, 41.04) mm, rotated rx 180 ry 0 rz 180 deg; joints [-38.269, -22.05, 85.788, 60.711, 45.246, -51.456]
  Call Extruder(57.87401)
  MoveL 1713 to (-39.05, 43.71, 41.04) mm, rotated rx 180 ry 0 rz -180 deg; joints [-38.207, -22.06, 85.793, 60.653, 45.199, -51.413]
  MoveL 1714 to (-39.05, 43.71, 41.04) mm, rotated rx 180 ry 0 rz -180 deg; joints [-38.207, -22.06, 85.793, 60.653, 45.199, -51.413]
  Call Extruder(58.03200)
  MoveL 1715 to (-38.94, 43.46, 41.04) mm, rotated rx 180 ry 0 rz 180 deg; joints [-38.149, -22.069, 85.798, 60.599, 45.156, -51.373]
  MoveL 1716 to (-38.94, 43.46, 41.04) mm, rotated rx 180 ry 0 rz 180 deg; joints [-38.149, -22.069, 85.798, 60.599, 45.156, -51.373]
  Call Extruder(58.19059)
  MoveL 1717 to (-38.84, 43.21, 41.04) mm, rotated rx 180 ry 0 rz 180 deg; joints [-38.092, -22.078, 85.804, 60.545, 45.113, -51.332]
  MoveL 1718 to (-38.84, 43.21, 41.04) mm, rotated rx 180 ry 0 rz 180 deg; joints [-38.092, -22.078, 85.804, 60.545, 45.113, -51.332]
  Call Extruder(58.39676)
  MoveL 1719 to (-38.66, 42.91, 41.04) mm, rotated rx 180 ry 0 rz 180 deg; joints [-38.016, -22.085, 85.807, 60.476, 45.055, -51.281]
  MoveL 1720 to (-38.66, 42.91, 41.04) mm, rotated rx 180 ry 0 rz 180 deg; joints [-38.016, -22.085, 85.807, 60.476, 45.055, -51.281]
  Call Extruder(58.60370)
  MoveL 1721 to (-38.49, 42.6, 41.04) mm, rotated rx 180 ry 0 rz 180 deg; joints [-37.939, -22.091, 85.811, 60.406, 44.997, -51.23]
  MoveL 1722 to (-38.49, 42.6, 41.04) mm, rotated rx 180 ry 0 rz 180 deg; joints [-37.939, -22.091, 85.811, 60.406, 44.997, -51.23]
  Call Extruder(58.81142)
  MoveL 1723 to (-38.31, 42.3, 41.04) mm, rotated rx -180 ry 0 rz 180 deg; joints [-37.863, -22.097, 85.814, 60.336, 44.939, -51.179]
  MoveL 1724 to (-38.31, 42.3, 41.04) mm, rotated rx -180 ry 0 rz 180 deg; joints [-37.863, -22.097, 85.814, 60.336, 44.939, -51.179]
  Call Extruder(59.01993)
  MoveL 1725 to (-38.13, 41.99, 41.04) mm, rotated rx 180 ry 0 rz 180 deg; joints [-37.787, -22.103, 85.818, 60.266, 44.88, -51.128]
  MoveL 1726 to (-38.13, 41.99, 41.04) mm, rotated rx 180 ry 0 rz 180 deg; joints [-37.787, -22.103, 85.818, 60.266, 44.88, -51.128]
  Call Extruder(59.19948)
  MoveL 1727 to (-37.96, 41.75, 41.04) mm, rotated rx 180 ry 0 rz 180 deg; joints [-37.72, -22.104, 85.819, 60.206, 44.829, -51.085]
  MoveL 1728 to (-37.96, 41.75, 41.04) mm, rotated rx 180 ry 0 rz 180 deg; joints [-37.72, -22.104, 85.819, 60.206, 44.829, -51.085]
  Call Extruder(59.53291)
  MoveL 1729 to (-37.63, 41.3, 41.04) mm, rotated rx 180 ry 0 rz 180 deg; joints [-37.598, -22.106, 85.82, 60.096, 44.734, -51.007]
  MoveL 1730 to (-37.63, 41.3, 41.04) mm, rotated rx 180 ry 0 rz 180 deg; joints [-37.598, -22.106, 85.82, 60.096, 44.734, -51.007]
  Call Extruder(59.86753)
  MoveL 1731 to (-37.3, 40.85, 41.04) mm, rotated rx 180 ry 0 rz 180 deg; joints [-37.475, -22.108, 85.821, 59.986, 44.639, -50.928]
  Call Extruder(60.69546)
  MoveL 1732 to (-36.39, 39.81, 41.04) mm, rotated rx -180 ry 0 rz 180 deg; joints [-37.173, -22.096, 85.814, 59.718, 44.402, -50.74]
  Call Extruder(61.52337)
  MoveL 1733 to (-35.35, 38.9, 41.04) mm, rotated rx 180 ry 0 rz 180 deg; joints [-36.876, -22.06, 85.793, 59.462, 44.165, -50.566]
  Call Extruder(61.69068)
  MoveL 1734 to (-35.13, 38.73, 41.04) mm, rotated rx 180 ry 0 rz 180 deg; joints [-36.818, -22.05, 85.787, 59.412, 44.118, -50.533]
  MoveL 1735 to (-35.13, 38.73, 41.04) mm, rotated rx 180 ry 0 rz 180 deg; joints [-36.818, -22.05, 85.787, 59.412, 44.118, -50.533]
  Call Extruder(62.02410)
  MoveL 1736 to (-34.68, 38.41, 41.03) mm, rotated rx 180 ry 0 rz -180 deg; joints [-36.701, -22.029, 85.775, 59.314, 44.023, -50.467]
  MoveL 1737 to (-34.68, 38.41, 41.03) mm, rotated rx 180 ry 0 rz -180 deg; joints [-36.701, -22.029, 85.775, 59.314, 44.023, -50.467]
  Call Extruder(62.35635)
  MoveL 1738 to (-34.23, 38.08, 41.04) mm, rotated rx -180 ry 0 rz 180 deg; joints [-36.584, -22.008, 85.763, 59.214, 43.928, -50.401]
  MoveL 1739 to (-34.23, 38.08, 41.04) mm, rotated rx -180 ry 0 rz 180 deg; joints [-36.584, -22.008, 85.763, 59.214, 43.928, -50.401]
  Call Extruder(62.47405)
  MoveL 1740 to (-34.05, 37.98, 41.03) mm, rotated rx -180 ry 0 rz -180 deg; joints [-36.544, -21.998, 85.757, 59.182, 43.896, -50.38]
  MoveL 1741 to (-34.05, 37.98, 41.03) mm, rotated rx -180 ry 0 rz -180 deg; joints [-36.544, -21.998, 85.757, 59.182, 43.896, -50.38]
  Call Extruder(62.68177)
  MoveL 1742 to (-33.75, 37.8, 41.04) mm, rotated rx 180 ry 0 rz 180 deg; joints [-36.474, -21.98, 85.747, 59.123, 43.837, -50.343]
  MoveL 1743 to (-33.75, 37.8, 41.04) mm, rotated rx 180 ry 0 rz 180 deg; joints [-36.474, -21.98, 85.747, 59.123, 43.837, -50.343]
  Call Extruder(62.88871)
  MoveL 1744 to (-33.45, 37.63, 41.04) mm, rotated rx 180 ry 0 rz 180 deg; joints [-36.403, -21.962, 85.736, 59.065, 43.779, -50.305]
  MoveL 1745 to (-33.45, 37.63, 41.04) mm, rotated rx 180 ry 0 rz 180 deg; joints [-36.403, -21.962, 85.736, 59.065, 43.779, -50.305]
  Call Extruder(63.09487)
  MoveL 1746 to (-33.14, 37.45, 41.04) mm, rotated rx 180 ry 0 rz -180 deg; joints [-36.333, -21.944, 85.726, 59.007, 43.722, -50.268]
  MoveL 1747 to (-33.14, 37.45, 41.04) mm, rotated rx 180 ry 0 rz -180 deg; joints [-36.333, -21.944, 85.726, 59.007, 43.722, -50.268]
  Call Extruder(63.27655)
  MoveL 1748 to (-32.87, 37.31, 41.04) mm, rotated rx 180 ry 0 rz 180 deg; joints [-36.272, -21.926, 85.716, 58.958, 43.671, -50.236]
  MoveL 1749 to (-32.87, 37.31, 41.04) mm, rotated rx 180 ry 0 rz 180 deg; joints [-36.272, -21.926, 85.716, 58.958, 43.671, -50.236]
  Call Extruder(63.43455)
  MoveL 1750 to (-32.62, 37.2, 41.03) mm, rotated rx -180 ry 0 rz 180 deg; joints [-36.221, -21.908, 85.705, 58.917, 43.628, -50.211]
  MoveL 1751 to (-32.62, 37.2, 41.03) mm, rotated rx -180 ry 0 rz 180 deg; joints [-36.221, -21.908, 85.705, 58.917, 43.628, -50.211]
  Call Extruder(63.59195)
  MoveL 1752 to (-32.37, 37.1, 41.04) mm, rotated rx 180 ry 0 rz 180 deg; joints [-36.17, -21.891, 85.695, 58.876, 43.585, -50.186]
  MoveL 1753 to (-32.37, 37.1, 41.04) mm, rotated rx 180 ry 0 rz 180 deg; joints [-36.17, -21.891, 85.695, 58.876, 43.585, -50.186]
  Call Extruder(63.77466)
  MoveL 1754 to (-32.08, 36.97, 41.04) mm, rotated rx 180 ry 0 rz 180 deg; joints [-36.112, -21.87, 85.683, 58.83, 43.535, -50.158]
  MoveL 1755 to (-32.08, 36.97, 41.04) mm, rotated rx 180 ry 0 rz 180 deg; joints [-36.112, -21.87, 85.683, 58.83, 43.535, -50.158]
  Call Extruder(63.95661)
  MoveL 1756 to (-31.78, 36.85, 41.04) mm, rotated rx 180 ry 0 rz 180 deg; joints [-36.053, -21.848, 85.671, 58.783, 43.485, -50.129]
  MoveL 1757 to (-31.78, 36.85, 41.04) mm, rotated rx 180 ry 0 rz 180 deg; joints [-36.053, -21.848, 85.671, 58.783, 43.485, -50.129]
  Call Extruder(64.10394)
  MoveL 1758 to (-31.54, 36.76, 41.03) mm, rotated rx 180 ry 0 rz 180 deg; joints [-36.006, -21.831, 85.66, 58.746, 43.446, -50.107]
  MoveL 1759 to (-31.54, 36.76, 41.03) mm, rotated rx 180 ry 0 rz 180 deg; joints [-36.006, -21.831, 85.66, 58.746, 43.446, -50.107]
  Call Extruder(64.21718)
  MoveL 1760 to (-31.35, 36.7, 41.04) mm, rotated rx 180 ry 0 rz 180 deg; joints [-35.971, -21.816, 85.652, 58.719, 43.415, -50.091]
  MoveL 1761 to (-31.35, 36.7, 41.04) mm, rotated rx 180 ry 0 rz 180 deg; joints [-35.971, -21.816, 85.652, 58.719, 43.415, -50.091]
  Call Extruder(64.32997)
  MoveL 1762 to (-31.17, 36.64, 41.04) mm, rotated rx 180 ry 0 rz 180 deg; joints [-35.936, -21.801, 85.643, 58.692, 43.386, -50.075]
  MoveL 1763 to (-31.17, 36.64, 41.04) mm, rotated rx 180 ry 0 rz 180 deg; joints [-35.936, -21.801, 85.643, 58.692, 43.386, -50.075]
  Call Extruder(64.44232)
  MoveL 1764 to (-30.98, 36.58, 41.04) mm, rotated rx 180 ry 0 rz -180 deg; joints [-35.901, -21.786, 85.634, 58.665, 43.356, -50.059]
  MoveL 1765 to (-30.98, 36.58, 41.04) mm, rotated rx 180 ry 0 rz -180 deg; joints [-35.901, -21.786, 85.634, 58.665, 43.356, -50.059]
  Call Extruder(64.55422)
  MoveL 1766 to (-30.79, 36.52, 41.04) mm, rotated rx 180 ry 0 rz 180 deg; joints [-35.867, -21.771, 85.626, 58.639, 43.326, -50.043]
  MoveL 1767 to (-30.79, 36.52, 41.04) mm, rotated rx 180 ry 0 rz 180 deg; joints [-35.867, -21.771, 85.626, 58.639, 43.326, -50.043]
  Call Extruder(64.67562)
  MoveL 1768 to (-30.58, 36.45, 41.04) mm, rotated rx 180 ry 0 rz 180 deg; joints [-35.829, -21.754, 85.616, 58.61, 43.293, -50.026]
  MoveL 1769 to (-30.58, 36.45, 41.04) mm, rotated rx 180 ry 0 rz 180 deg; joints [-35.829, -21.754, 85.616, 58.61, 43.293, -50.026]
  Call Extruder(64.80641)
  MoveL 1770 to (-30.36, 36.38, 41.04) mm, rotated rx 180 ry 0 rz 180 deg; joints [-35.788, -21.736, 85.605, 58.579, 43.258, -50.008]
  MoveL 1771 to (-30.36, 36.38, 41.04) mm, rotated rx 180 ry 0 rz 180 deg; joints [-35.788, -21.736, 85.605, 58.579, 43.258, -50.008]
  Call Extruder(64.93664)
  MoveL 1772 to (-30.14, 36.32, 41.04) mm, rotated rx 180 ry 0 rz -180 deg; joints [-35.748, -21.718, 85.595, 58.548, 43.224, -49.99]
  MoveL 1773 to (-30.14, 36.32, 41.04) mm, rotated rx 180 ry 0 rz -180 deg; joints [-35.748, -21.718, 85.595, 58.548, 43.224, -49.99]
  Call Extruder(65.06630)
  MoveL 1774 to (-29.91, 36.25, 41.04) mm, rotated rx 180 ry 0 rz 180 deg; joints [-35.708, -21.7, 85.584, 58.517, 43.189, -49.972]
  MoveL 1775 to (-29.91, 36.25, 41.04) mm, rotated rx 180 ry 0 rz 180 deg; joints [-35.708, -21.7, 85.584, 58.517, 43.189, -49.972]
  Call Extruder(65.19540)
  MoveL 1776 to (-29.69, 36.18, 41.04) mm, rotated rx 180 ry 0 rz 180 deg; joints [-35.668, -21.681, 85.573, 58.486, 43.154, -49.954]
  MoveL 1777 to (-29.69, 36.18, 41.04) mm, rotated rx 180 ry 0 rz 180 deg; joints [-35.668, -21.681, 85.573, 58.486, 43.154, -49.954]
  Call Extruder(65.31047)
  MoveL 1778 to (-29.48, 36.14, 41.04) mm, rotated rx 180 ry 0 rz 180 deg; joints [-35.634, -21.663, 85.563, 58.461, 43.124, -49.94]
  MoveL 1779 to (-29.48, 36.14, 41.04) mm, rotated rx 180 ry 0 rz 180 deg; joints [-35.634, -21.663, 85.563, 58.461, 43.124, -49.94]
  Call Extruder(65.42509)
  MoveL 1780 to (-29.28, 36.09, 41.04) mm, rotated rx -180 ry 0 rz 180 deg; joints [-35.601, -21.646, 85.553, 58.436, 43.095, -49.926]
  MoveL 1781 to (-29.28, 36.09, 41.04) mm, rotated rx -180 ry 0 rz 180 deg; joints [-35.601, -21.646, 85.553, 58.436, 43.095, -49.926]
  Call Extruder(65.53926)
  MoveL 1782 to (-29.08, 36.05, 41.04) mm, rotated rx 180 ry 0 rz 180 deg; joints [-35.567, -21.628, 85.542, 58.411, 43.065, -49.912]
  MoveL 1783 to (-29.08, 36.05, 41.04) mm, rotated rx 180 ry 0 rz 180 deg; joints [-35.567, -21.628, 85.542, 58.411, 43.065, -49.912]
  Call Extruder(65.65298)
  MoveL 1784 to (-28.87, 36, 41.04) mm, rotated rx -180 ry 0 rz -180 deg; joints [-35.533, -21.61, 85.531, 58.386, 43.035, -49.899]
  MoveL 1785 to (-28.87, 36, 41.04) mm, rotated rx -180 ry 0 rz -180 deg; joints [-35.533, -21.61, 85.531, 58.386, 43.035, -49.899]
  Call Extruder(65.77840)
  MoveL 1786 to (-28.64, 35.96, 41.04) mm, rotated rx 180 ry 0 rz 180 deg; joints [-35.497, -21.589, 85.52, 58.359, 43.003, -49.884]
  MoveL 1787 to (-28.64, 35.96, 41.04) mm, rotated rx 180 ry 0 rz 180 deg; joints [-35.497, -21.589, 85.52, 58.359, 43.003, -49.884]
  Call Extruder(65.91538)
  MoveL 1788 to (-28.4, 35.91, 41.04) mm, rotated rx 180 ry 0 rz 180 deg; joints [-35.457, -21.567, 85.507, 58.33, 42.968, -49.867]
  MoveL 1789 to (-28.4, 35.91, 41.04) mm, rotated rx 180 ry 0 rz 180 deg; joints [-35.457, -21.567, 85.507, 58.33, 42.968, -49.867]
  Call Extruder(66.05174)
  MoveL 1790 to (-28.15, 35.86, 41.04) mm, rotated rx 180 ry 0 rz 180 deg; joints [-35.417, -21.545, 85.493, 58.301, 42.932, -49.851]
  MoveL 1791 to (-28.15, 35.86, 41.04) mm, rotated rx 180 ry 0 rz 180 deg; joints [-35.417, -21.545, 85.493, 58.301, 42.932, -49.851]
  Call Extruder(66.18750)
  MoveL 1792 to (-27.9, 35.81, 41.04) mm, rotated rx -180 ry 0 rz 180 deg; joints [-35.377, -21.522, 85.48, 58.271, 42.897, -49.835]
  MoveL 1793 to (-27.9, 35.81, 41.04) mm, rotated rx -180 ry 0 rz 180 deg; joints [-35.377, -21.522, 85.48, 58.271, 42.897, -49.835]
  Call Extruder(66.32265)
  MoveL 1794 to (-27.65, 35.76, 41.04) mm, rotated rx -180 ry 0 rz 180 deg; joints [-35.337, -21.5, 85.467, 58.242, 42.862, -49.819]
  MoveL 1795 to (-27.65, 35.76, 41.04) mm, rotated rx -180 ry 0 rz 180 deg; joints [-35.337, -21.5, 85.467, 58.242, 42.862, -49.819]
  Call Extruder(66.45718)
  MoveL 1796 to (-27.4, 35.71, 41.04) mm, rotated rx -180 ry 0 rz -180 deg; joints [-35.297, -21.478, 85.454, 58.213, 42.826, -49.803]
  MoveL 1797 to (-27.4, 35.71, 41.04) mm, rotated rx -180 ry 0 rz -180 deg; joints [-35.297, -21.478, 85.454, 58.213, 42.826, -49.803]
  Call Extruder(66.59111)
  MoveL 1798 to (-27.15, 35.66, 41.03) mm, rotated rx -180 ry 0 rz 180 deg; joints [-35.258, -21.455, 85.441, 58.184, 42.791, -49.787]
  MoveL 1799 to (-27.15, 35.66, 41.03) mm, rotated rx -180 ry 0 rz 180 deg; joints [-35.258, -21.455, 85.441, 58.184, 42.791, -49.787]
  Call Extruder(66.73897)
  MoveL 1800 to (-26.87, 35.61, 41.04) mm, rotated rx -180 ry 0 rz -180 deg; joints [-35.215, -21.43, 85.426, 58.152, 42.753, -49.77]
  MoveL 1801 to (-26.87, 35.61, 41.04) mm, rotated rx -180 ry 0 rz -180 deg; joints [-35.215, -21.43, 85.426, 58.152, 42.753, -49.77]
  Call Extruder(66.90071)
  MoveL 1802 to (-26.57, 35.56, 41.04) mm, rotated rx 180 ry 0 rz 180 deg; joints [-35.168, -21.401, 85.409, 58.119, 42.711, -49.752]
  MoveL 1803 to (-26.57, 35.56, 41.04) mm, rotated rx 180 ry 0 rz 180 deg; joints [-35.168, -21.401, 85.409, 58.119, 42.711, -49.752]
  Call Extruder(67.06171)
  MoveL 1804 to (-26.26, 35.51, 41.04) mm, rotated rx -180 ry 0 rz 180 deg; joints [-35.122, -21.372, 85.392, 58.085, 42.67, -49.734]
  MoveL 1805 to (-26.26, 35.51, 41.04) mm, rotated rx -180 ry 0 rz 180 deg; joints [-35.122, -21.372, 85.392, 58.085, 42.67, -49.734]
  Call Extruder(67.22199)
  MoveL 1806 to (-25.96, 35.47, 41.03) mm, rotated rx 180 ry 0 rz 180 deg; joints [-35.075, -21.344, 85.375, 58.052, 42.628, -49.716]
  MoveL 1807 to (-25.96, 35.47, 41.03) mm, rotated rx 180 ry 0 rz 180 deg; joints [-35.075, -21.344, 85.375, 58.052, 42.628, -49.716]
  Call Extruder(67.38154)
  MoveL 1808 to (-25.65, 35.42, 41.04) mm, rotated rx 180 ry 0 rz 180 deg; joints [-35.029, -21.315, 85.358, 58.019, 42.587, -49.699]
  MoveL 1809 to (-25.65, 35.42, 41.04) mm, rotated rx 180 ry 0 rz 180 deg; joints [-35.029, -21.315, 85.358, 58.019, 42.587, -49.699]
  Call Extruder(67.54036)
  MoveL 1810 to (-25.34, 35.37, 41.04) mm, rotated rx 180 ry 0 rz 180 deg; joints [-34.983, -21.287, 85.341, 57.985, 42.545, -49.681]
  MoveL 1811 to (-25.34, 35.37, 41.04) mm, rotated rx 180 ry 0 rz 180 deg; joints [-34.983, -21.287, 85.341, 57.985, 42.545, -49.681]
  Call Extruder(67.71903)
  MoveL 1812 to (-25, 35.32, 41.03) mm, rotated rx 180 ry 0 rz 180 deg; joints [-34.932, -21.254, 85.322, 57.949, 42.499, -49.662]
  MoveL 1813 to (-25, 35.32, 41.03) mm, rotated rx 180 ry 0 rz 180 deg; joints [-34.932, -21.254, 85.322, 57.949, 42.499, -49.662]
  Call Extruder(67.91748)
  MoveL 1814 to (-24.61, 35.28, 41.04) mm, rotated rx 180 ry 0 rz 180 deg; joints [-34.877, -21.216, 85.3, 57.91, 42.449, -49.642]
  MoveL 1815 to (-24.61, 35.28, 41.04) mm, rotated rx 180 ry 0 rz 180 deg; joints [-34.877, -21.216, 85.3, 57.91, 42.449, -49.642]
  Call Extruder(68.11505)
  MoveL 1816 to (-24.22, 35.23, 41.04) mm, rotated rx 180 ry 0 rz 180 deg; joints [-34.821, -21.179, 85.277, 57.871, 42.399, -49.622]
  MoveL 1817 to (-24.22, 35.23, 41.04) mm, rotated rx 180 ry 0 rz 180 deg; joints [-34.821, -21.179, 85.277, 57.871, 42.399, -49.622]
  Call Extruder(68.31176)
  MoveL 1818 to (-23.84, 35.18, 41.04) mm, rotated rx -180 ry 0 rz 180 deg; joints [-34.766, -21.141, 85.255, 57.832, 42.348, -49.602]
  MoveL 1819 to (-23.84, 35.18, 41.04) mm, rotated rx -180 ry 0 rz 180 deg; joints [-34.766, -21.141, 85.255, 57.832, 42.348, -49.602]
  Call Extruder(68.50760)
  MoveL 1820 to (-23.45, 35.14, 41.04) mm, rotated rx 180 ry 0 rz -180 deg; joints [-34.711, -21.103, 85.232, 57.793, 42.298, -49.582]
  MoveL 1821 to (-23.45, 35.14, 41.04) mm, rotated rx 180 ry 0 rz -180 deg; joints [-34.711, -21.103, 85.232, 57.793, 42.298, -49.582]
  Call Extruder(68.80299)
  MoveL 1822 to (-22.86, 35.09, 41.04) mm, rotated rx 180 ry 0 rz 180 deg; joints [-34.631, -21.044, 85.197, 57.738, 42.225, -49.555]
  MoveL 1823 to (-22.86, 35.09, 41.04) mm, rotated rx 180 ry 0 rz 180 deg; joints [-34.631, -21.044, 85.197, 57.738, 42.225, -49.555]
  Call Extruder(69.09705)
  MoveL 1824 to (-22.27, 35.04, 41.04) mm, rotated rx -180 ry 0 rz 180 deg; joints [-34.552, -20.985, 85.162, 57.684, 42.152, -49.528]
  MoveL 1825 to (-22.27, 35.04, 41.04) mm, rotated rx -180 ry 0 rz 180 deg; joints [-34.552, -20.985, 85.162, 57.684, 42.152, -49.528]
  Call Extruder(69.38978)
  MoveL 1826 to (-21.68, 35, 41.04) mm, rotated rx -180 ry 0 rz 180 deg; joints [-34.473, -20.926, 85.126, 57.63, 42.079, -49.501]
  MoveL 1827 to (-21.68, 35, 41.04) mm, rotated rx -180 ry 0 rz 180 deg; joints [-34.473, -20.926, 85.126, 57.63, 42.079, -49.501]
  Call Extruder(69.96323)
  MoveL 1828 to (-20.52, 34.95, 41.04) mm, rotated rx 180 ry 0 rz 180 deg; joints [-34.326, -20.805, 85.054, 57.532, 41.942, -49.456]
  MoveL 1829 to (-20.52, 34.95, 41.04) mm, rotated rx 180 ry 0 rz 180 deg; joints [-34.326, -20.805, 85.054, 57.532, 41.942, -49.456]
  Call Extruder(70.67720)
  MoveL 1830 to (-19.06, 34.91, 41.04) mm, rotated rx 180 ry 0 rz 180 deg; joints [-34.146, -20.653, 84.962, 57.414, 41.773, -49.402]
  Call Extruder(187.52394)
  MoveL 1831 to (219.06, 34.91, 41.03) mm, rotated rx 180 ry 0 rz 180 deg; joints [-18.248, 11.905, 55.099, 40.163, 29.046, -36.421]
  Call Extruder(187.95250)
  MoveL 1832 to (219.94, 34.93, 41.04) mm, rotated rx 180 ry 0 rz 180 deg; joints [-18.218, 12.063, 54.905, 40.072, 29.055, -36.33]
  MoveL 1833 to (219.94, 34.93, 41.04) mm, rotated rx 180 ry 0 rz 180 deg; joints [-18.218, 12.063, 54.905, 40.072, 29.055, -36.33]
  Call Extruder(188.52594)
  MoveL 1834 to (221.1, 34.98, 41.03) mm, rotated rx 180 ry 0 rz 180 deg; joints [-18.181, 12.275, 54.645, 39.954, 29.07, -36.212]
  MoveL 1835 to (221.1, 34.98, 41.03) mm, rotated rx 180 ry 0 rz 180 deg; joints [-18.181, 12.275, 54.645, 39.954, 29.07, -36.212]
  Call Extruder(188.96026)
  MoveL 1836 to (221.97, 35.02, 41.03) mm, rotated rx 180 ry 0 rz 180 deg; joints [-18.154, 12.436, 54.446, 39.867, 29.083, -36.124]
  MoveL 1837 to (221.97, 35.02, 41.03) mm, rotated rx 180 ry 0 rz 180 deg; joints [-18.154, 12.436, 54.446, 39.867, 29.083, -36.124]
  Call Extruder(189.25431)
  MoveL 1838 to (222.56, 35.07, 41.04) mm, rotated rx -180 ry 0 rz 180 deg; joints [-18.138, 12.546, 54.31, 39.81, 29.093, -36.066]
  MoveL 1839 to (222.56, 35.07, 41.04) mm, rotated rx -180 ry 0 rz 180 deg; joints [-18.138, 12.546, 54.31, 39.81, 29.093, -36.066]
  Call Extruder(189.54970)
  MoveL 1840 to (223.15, 35.11, 41.04) mm, rotated rx 180 ry 0 rz -180 deg; joints [-18.121, 12.656, 54.174, 39.753, 29.103, -36.008]
  MoveL 1841 to (223.15, 35.11, 41.04) mm, rotated rx 180 ry 0 rz -180 deg; joints [-18.121, 12.656, 54.174, 39.753, 29.103, -36.008]
  Call Extruder(189.79594)
  MoveL 1842 to (223.64, 35.16, 41.04) mm, rotated rx -180 ry 0 rz 180 deg; joints [-18.109, 12.748, 54.06, 39.707, 29.113, -35.961]
  MoveL 1843 to (223.64, 35.16, 41.04) mm, rotated rx -180 ry 0 rz 180 deg; joints [-18.109, 12.748, 54.06, 39.707, 29.113, -35.961]
  Call Extruder(189.99264)
  MoveL 1844 to (224.03, 35.21, 41.04) mm, rotated rx -180 ry 0 rz 180 deg; joints [-18.1, 12.822, 53.969, 39.672, 29.121, -35.925]
  MoveL 1845 to (224.03, 35.21, 41.04) mm, rotated rx -180 ry 0 rz 180 deg; joints [-18.1, 12.822, 53.969, 39.672, 29.121, -35.925]
  Call Extruder(190.19022)
  MoveL 1846 to (224.42, 35.25, 41.04) mm, rotated rx 180 ry 0 rz 180 deg; joints [-18.091, 12.896, 53.878, 39.637, 29.129, -35.889]
  MoveL 1847 to (224.42, 35.25, 41.04) mm, rotated rx 180 ry 0 rz 180 deg; joints [-18.091, 12.896, 53.878, 39.637, 29.129, -35.889]
  Call Extruder(190.38866)
  MoveL 1848 to (224.8, 35.3, 41.04) mm, rotated rx -180 ry 0 rz 180 deg; joints [-18.082, 12.97, 53.786, 39.601, 29.138, -35.852]
  MoveL 1849 to (224.8, 35.3, 41.04) mm, rotated rx -180 ry 0 rz 180 deg; joints [-18.082, 12.97, 53.786, 39.601, 29.138, -35.852]
  Call Extruder(190.58797)
  MoveL 1850 to (225.19, 35.34, 41.04) mm, rotated rx -180 ry 0 rz 180 deg; joints [-18.073, 13.043, 53.694, 39.566, 29.147, -35.816]
  MoveL 1851 to (225.19, 35.34, 41.04) mm, rotated rx -180 ry 0 rz 180 deg; joints [-18.073, 13.043, 53.694, 39.566, 29.147, -35.816]
  Call Extruder(190.74679)
  MoveL 1852 to (225.5, 35.39, 41.04) mm, rotated rx -180 ry 0 rz -180 deg; joints [-18.068, 13.103, 53.62, 39.54, 29.155, -35.789]
  MoveL 1853 to (225.5, 35.39, 41.04) mm, rotated rx -180 ry 0 rz -180 deg; joints [-18.068, 13.103, 53.62, 39.54, 29.155, -35.789]
  Call Extruder(190.90634)
  MoveL 1854 to (225.8, 35.44, 41.04) mm, rotated rx -180 ry 0 rz 180 deg; joints [-18.062, 13.162, 53.546, 39.514, 29.163, -35.761]
  MoveL 1855 to (225.8, 35.44, 41.04) mm, rotated rx -180 ry 0 rz 180 deg; joints [-18.062, 13.162, 53.546, 39.514, 29.163, -35.761]
  Call Extruder(191.06662)
  MoveL 1856 to (226.11, 35.49, 41.04) mm, rotated rx 180 ry 0 rz 180 deg; joints [-18.056, 13.221, 53.472, 39.488, 29.171, -35.734]
  MoveL 1857 to (226.11, 35.49, 41.04) mm, rotated rx 180 ry 0 rz 180 deg; joints [-18.056, 13.221, 53.472, 39.488, 29.171, -35.734]
  Call Extruder(191.22762)
  MoveL 1858 to (226.41, 35.54, 41.04) mm, rotated rx -180 ry 0 rz 180 deg; joints [-18.051, 13.281, 53.398, 39.462, 29.179, -35.707]
  MoveL 1859 to (226.41, 35.54, 41.04) mm, rotated rx -180 ry 0 rz 180 deg; joints [-18.051, 13.281, 53.398, 39.462, 29.179, -35.707]
  Call Extruder(191.38936)
  MoveL 1860 to (226.72, 35.59, 41.04) mm, rotated rx 180 ry 0 rz 180 deg; joints [-18.045, 13.34, 53.324, 39.435, 29.187, -35.679]
  MoveL 1861 to (226.72, 35.59, 41.04) mm, rotated rx 180 ry 0 rz 180 deg; joints [-18.045, 13.34, 53.324, 39.435, 29.187, -35.679]
  Call Extruder(191.55182)
  MoveL 1862 to (227.03, 35.64, 41.04) mm, rotated rx 180 ry 0 rz 180 deg; joints [-18.039, 13.4, 53.249, 39.409, 29.195, -35.651]
  MoveL 1863 to (227.03, 35.64, 41.04) mm, rotated rx 180 ry 0 rz 180 deg; joints [-18.039, 13.4, 53.249, 39.409, 29.195, -35.651]
  Call Extruder(191.68574)
  MoveL 1864 to (227.28, 35.68, 41.04) mm, rotated rx -180 ry 0 rz 180 deg; joints [-18.036, 13.449, 53.188, 39.389, 29.203, -35.63]
  MoveL 1865 to (227.28, 35.68, 41.04) mm, rotated rx -180 ry 0 rz 180 deg; joints [-18.036, 13.449, 53.188, 39.389, 29.203, -35.63]
  Call Extruder(191.82028)
  MoveL 1866 to (227.52, 35.73, 41.03) mm, rotated rx -180 ry 0 rz 180 deg; joints [-18.033, 13.498, 53.126, 39.369, 29.21, -35.609]
  MoveL 1867 to (227.52, 35.73, 41.03) mm, rotated rx -180 ry 0 rz 180 deg; joints [-18.033, 13.498, 53.126, 39.369, 29.21, -35.609]
  Call Extruder(191.95543)
  MoveL 1868 to (227.77, 35.78, 41.04) mm, rotated rx 180 ry 0 rz 180 deg; joints [-18.029, 13.547, 53.064, 39.349, 29.218, -35.588]
  MoveL 1869 to (227.77, 35.78, 41.04) mm, rotated rx 180 ry 0 rz 180 deg; joints [-18.029, 13.547, 53.064, 39.349, 29.218, -35.588]
  Call Extruder(192.09119)
  MoveL 1870 to (228.02, 35.83, 41.04) mm, rotated rx -180 ry 0 rz 180 deg; joints [-18.026, 13.597, 53.002, 39.329, 29.226, -35.566]
  MoveL 1871 to (228.02, 35.83, 41.04) mm, rotated rx -180 ry 0 rz 180 deg; joints [-18.026, 13.597, 53.002, 39.329, 29.226, -35.566]
  Call Extruder(192.22756)
  MoveL 1872 to (228.27, 35.88, 41.04) mm, rotated rx -180 ry 0 rz 180 deg; joints [-18.022, 13.646, 52.94, 39.309, 29.234, -35.545]
  MoveL 1873 to (228.27, 35.88, 41.04) mm, rotated rx -180 ry 0 rz 180 deg; joints [-18.022, 13.646, 52.94, 39.309, 29.234, -35.545]
  Call Extruder(192.36453)
  MoveL 1874 to (228.52, 35.93, 41.04) mm, rotated rx 180 ry 0 rz 180 deg; joints [-18.019, 13.696, 52.878, 39.289, 29.241, -35.523]
  MoveL 1875 to (228.52, 35.93, 41.04) mm, rotated rx 180 ry 0 rz 180 deg; joints [-18.019, 13.696, 52.878, 39.289, 29.241, -35.523]
  Call Extruder(192.50212)
  MoveL 1876 to (228.77, 35.98, 41.04) mm, rotated rx -180 ry 0 rz 180 deg; joints [-18.015, 13.745, 52.816, 39.269, 29.249, -35.502]
  MoveL 1877 to (228.77, 35.98, 41.04) mm, rotated rx -180 ry 0 rz 180 deg; joints [-18.015, 13.745, 52.816, 39.269, 29.249, -35.502]
  Call Extruder(192.61584)
  MoveL 1878 to (228.97, 36.03, 41.04) mm, rotated rx -180 ry 0 rz -180 deg; joints [-18.013, 13.786, 52.764, 39.253, 29.256, -35.485]
  MoveL 1879 to (228.97, 36.03, 41.04) mm, rotated rx -180 ry 0 rz -180 deg; joints [-18.013, 13.786, 52.764, 39.253, 29.256, -35.485]
  Call Extruder(192.73001)
  MoveL 1880 to (229.18, 36.07, 41.04) mm, rotated rx -180 ry 0 rz 180 deg; joints [-18.01, 13.827, 52.713, 39.237, 29.263, -35.467]
  MoveL 1881 to (229.18, 36.07, 41.04) mm, rotated rx -180 ry 0 rz 180 deg; joints [-18.01, 13.827, 52.713, 39.237, 29.263, -35.467]
  Call Extruder(192.84463)
  MoveL 1882 to (229.38, 36.12, 41.04) mm, rotated rx 180 ry 0 rz 180 deg; joints [-18.008, 13.868, 52.661, 39.221, 29.27, -35.45]
  MoveL 1883 to (229.38, 36.12, 41.04) mm, rotated rx 180 ry 0 rz 180 deg; joints [-18.008, 13.868, 52.661, 39.221, 29.27, -35.45]
  Call Extruder(192.95971)
  MoveL 1884 to (229.59, 36.16, 41.04) mm, rotated rx 180 ry 0 rz 180 deg; joints [-18.006, 13.909, 52.609, 39.205, 29.277, -35.433]
  MoveL 1885 to (229.59, 36.16, 41.04) mm, rotated rx 180 ry 0 rz 180 deg; joints [-18.006, 13.909, 52.609, 39.205, 29.277, -35.433]
  Call Extruder(193.08194)
  MoveL 1886 to (229.8, 36.22, 41.04) mm, rotated rx 180 ry 0 rz 180 deg; joints [-18.004, 13.952, 52.554, 39.189, 29.285, -35.416]
  MoveL 1887 to (229.8, 36.22, 41.04) mm, rotated rx 180 ry 0 rz 180 deg; joints [-18.004, 13.952, 52.554, 39.189, 29.285, -35.416]
  Call Extruder(193.21160)
  MoveL 1888 to (230.02, 36.28, 41.04) mm, rotated rx -180 ry 0 rz 180 deg; joints [-18.004, 13.999, 52.496, 39.175, 29.294, -35.4]
  MoveL 1889 to (230.02, 36.28, 41.04) mm, rotated rx -180 ry 0 rz 180 deg; joints [-18.004, 13.999, 52.496, 39.175, 29.294, -35.4]
  Call Extruder(193.34183)
  MoveL 1890 to (230.25, 36.35, 41.04) mm, rotated rx 180 ry 0 rz 180 deg; joints [-18.003, 14.045, 52.438, 39.16, 29.303, -35.383]
  MoveL 1891 to (230.25, 36.35, 41.04) mm, rotated rx 180 ry 0 rz 180 deg; joints [-18.003, 14.045, 52.438, 39.16, 29.303, -35.383]
  Call Extruder(193.47263)
  MoveL 1892 to (230.47, 36.42, 41.03) mm, rotated rx 180 ry 0 rz 180 deg; joints [-18.003, 14.091, 52.379, 39.146, 29.312, -35.366]
  MoveL 1893 to (230.47, 36.42, 41.03) mm, rotated rx 180 ry 0 rz 180 deg; joints [-18.003, 14.091, 52.379, 39.146, 29.312, -35.366]
  Call Extruder(193.60399)
  MoveL 1894 to (230.69, 36.49, 41.04) mm, rotated rx -180 ry 0 rz 180 deg; joints [-18.002, 14.137, 52.321, 39.131, 29.321, -35.35]
  MoveL 1895 to (230.69, 36.49, 41.04) mm, rotated rx -180 ry 0 rz 180 deg; joints [-18.002, 14.137, 52.321, 39.131, 29.321, -35.35]
  Call Extruder(193.72432)
  MoveL 1896 to (230.9, 36.55, 41.04) mm, rotated rx 180 ry 0 rz 180 deg; joints [-18.002, 14.18, 52.267, 39.118, 29.33, -35.335]
  MoveL 1897 to (230.9, 36.55, 41.04) mm, rotated rx 180 ry 0 rz 180 deg; joints [-18.002, 14.18, 52.267, 39.118, 29.33, -35.335]
  Call Extruder(193.84516)
  MoveL 1898 to (231.1, 36.62, 41.03) mm, rotated rx 180 ry 0 rz -180 deg; joints [-18.002, 14.222, 52.213, 39.106, 29.339, -35.321]
  MoveL 1899 to (231.1, 36.62, 41.03) mm, rotated rx 180 ry 0 rz -180 deg; joints [-18.002, 14.222, 52.213, 39.106, 29.339, -35.321]
  Call Extruder(193.96651)
  MoveL 1900 to (231.3, 36.68, 41.04) mm, rotated rx 180 ry 0 rz 180 deg; joints [-18.002, 14.264, 52.16, 39.093, 29.348, -35.306]
  MoveL 1901 to (231.3, 36.68, 41.04) mm, rotated rx 180 ry 0 rz 180 deg; joints [-18.002, 14.264, 52.16, 39.093, 29.348, -35.306]
  Call Extruder(194.08838)
  MoveL 1902 to (231.5, 36.75, 41.04) mm, rotated rx -180 ry 0 rz 180 deg; joints [-18.002, 14.307, 52.106, 39.08, 29.356, -35.292]
  MoveL 1903 to (231.5, 36.75, 41.04) mm, rotated rx -180 ry 0 rz 180 deg; joints [-18.002, 14.307, 52.106, 39.08, 29.356, -35.292]
  Call Extruder(194.21076)
  MoveL 1904 to (231.71, 36.82, 41.04) mm, rotated rx -180 ry 0 rz 180 deg; joints [-18.002, 14.349, 52.052, 39.067, 29.365, -35.277]
  MoveL 1905 to (231.71, 36.82, 41.04) mm, rotated rx -180 ry 0 rz 180 deg; joints [-18.002, 14.349, 52.052, 39.067, 29.365, -35.277]
  Call Extruder(194.33365)
  MoveL 1906 to (231.91, 36.88, 41.04) mm, rotated rx 180 ry 0 rz 180 deg; joints [-18.002, 14.391, 51.998, 39.055, 29.374, -35.262]
  MoveL 1907 to (231.91, 36.88, 41.04) mm, rotated rx 180 ry 0 rz 180 deg; joints [-18.002, 14.391, 51.998, 39.055, 29.374, -35.262]
  Call Extruder(194.51082)
  MoveL 1908 to (232.19, 37, 41.04) mm, rotated rx 180 ry 0 rz 180 deg; joints [-18.005, 14.452, 51.921, 39.041, 29.389, -35.245]
  MoveL 1909 to (232.19, 37, 41.04) mm, rotated rx 180 ry 0 rz 180 deg; joints [-18.005, 14.452, 51.921, 39.041, 29.389, -35.245]
  Call Extruder(194.72368)
  MoveL 1910 to (232.53, 37.15, 41.04) mm, rotated rx 180 ry 0 rz 180 deg; joints [-18.01, 14.525, 51.828, 39.026, 29.407, -35.226]
  MoveL 1911 to (232.53, 37.15, 41.04) mm, rotated rx 180 ry 0 rz 180 deg; joints [-18.01, 14.525, 51.828, 39.026, 29.407, -35.226]
  Call Extruder(194.91775)
  MoveL 1912 to (232.83, 37.29, 41.04) mm, rotated rx 180 ry 0 rz 180 deg; joints [-18.014, 14.591, 51.744, 39.013, 29.423, -35.209]
  MoveL 1913 to (232.83, 37.29, 41.04) mm, rotated rx 180 ry 0 rz 180 deg; joints [-18.014, 14.591, 51.744, 39.013, 29.423, -35.209]
  Call Extruder(195.11861)
  MoveL 1914 to (233.13, 37.45, 41.04) mm, rotated rx 180 ry 0 rz 180 deg; joints [-18.02, 14.659, 51.658, 39.003, 29.441, -35.195]
  MoveL 1915 to (233.13, 37.45, 41.04) mm, rotated rx 180 ry 0 rz 180 deg; joints [-18.02, 14.659, 51.658, 39.003, 29.441, -35.195]
  Call Extruder(195.32676)
  MoveL 1916 to (233.44, 37.62, 41.04) mm, rotated rx -180 ry 0 rz 180 deg; joints [-18.029, 14.729, 51.569, 38.995, 29.461, -35.182]
  MoveL 1917 to (233.44, 37.62, 41.04) mm, rotated rx -180 ry 0 rz 180 deg; joints [-18.029, 14.729, 51.569, 38.995, 29.461, -35.182]
  Call Extruder(195.53571)
  MoveL 1918 to (233.75, 37.8, 41.03) mm, rotated rx 180 ry 0 rz -180 deg; joints [-18.037, 14.798, 51.48, 38.988, 29.481, -35.169]
  MoveL 1919 to (233.75, 37.8, 41.03) mm, rotated rx 180 ry 0 rz -180 deg; joints [-18.037, 14.798, 51.48, 38.988, 29.481, -35.169]
  Call Extruder(195.74544)
  MoveL 1920 to (234.05, 37.98, 41.03) mm, rotated rx 180 ry 0 rz -180 deg; joints [-18.045, 14.868, 51.391, 38.98, 29.501, -35.156]
  MoveL 1921 to (234.05, 37.98, 41.03) mm, rotated rx 180 ry 0 rz -180 deg; joints [-18.045, 14.868, 51.391, 38.98, 29.501, -35.156]
  Call Extruder(195.86398)
  MoveL 1922 to (234.23, 38.08, 41.03) mm, rotated rx 180 ry 0 rz 180 deg; joints [-18.05, 14.907, 51.34, 38.975, 29.512, -35.149]
  MoveL 1923 to (234.23, 38.08, 41.03) mm, rotated rx 180 ry 0 rz 180 deg; joints [-18.05, 14.907, 51.34, 38.975, 29.512, -35.149]
  Call Extruder(196.19680)
  MoveL 1924 to (234.68, 38.41, 41.04) mm, rotated rx 180 ry 0 rz 180 deg; joints [-18.07, 15.015, 51.202, 38.974, 29.547, -35.139]
  MoveL 1925 to (234.68, 38.41, 41.04) mm, rotated rx 180 ry 0 rz 180 deg; joints [-18.07, 15.015, 51.202, 38.974, 29.547, -35.139]
  Call Extruder(196.53081)
  MoveL 1926 to (235.13, 38.73, 41.04) mm, rotated rx -180 ry 0 rz 180 deg; joints [-18.089, 15.122, 51.064, 38.973, 29.582, -35.128]
  MoveL 1927 to (235.13, 38.73, 41.04) mm, rotated rx -180 ry 0 rz 180 deg; joints [-18.089, 15.122, 51.064, 38.973, 29.582, -35.128]
  Call Extruder(196.69838)
  MoveL 1928 to (235.35, 38.9, 41.03) mm, rotated rx 180 ry 0 rz 180 deg; joints [-18.099, 15.176, 50.995, 38.972, 29.6, -35.123]
  Call Extruder(197.52772)
  MoveL 1929 to (236.39, 39.81, 41.04) mm, rotated rx -180 ry 0 rz 180 deg; joints [-18.16, 15.435, 50.662, 38.991, 29.693, -35.116]
  Call Extruder(198.15878)
  MoveL 1930 to (237.09, 40.59, 41.04) mm, rotated rx 180 ry 0 rz 180 deg; joints [-18.22, 15.621, 50.421, 39.03, 29.77, -35.133]
  MoveL 1931 to (237.09, 40.59, 41.04) mm, rotated rx 180 ry 0 rz 180 deg; joints [-18.22, 15.621, 50.421, 39.03, 29.77, -35.133]
  Call Extruder(198.35639)
  MoveL 1932 to (237.3, 40.85, 41.04) mm, rotated rx 180 ry 0 rz 180 deg; joints [-18.24, 15.679, 50.346, 39.043, 29.794, -35.139]
  Call Extruder(198.69040)
  MoveL 1933 to (237.63, 41.3, 41.03) mm, rotated rx 180 ry 0 rz 180 deg; joints [-18.277, 15.773, 50.225, 39.073, 29.837, -35.156]
  MoveL 1934 to (237.63, 41.3, 41.03) mm, rotated rx 180 ry 0 rz 180 deg; joints [-18.277, 15.773, 50.225, 39.073, 29.837, -35.156]
  Call Extruder(199.02322)
  MoveL 1935 to (237.96, 41.75, 41.04) mm, rotated rx 180 ry 0 rz 180 deg; joints [-18.313, 15.866, 50.103, 39.103, 29.88, -35.173]
  MoveL 1936 to (237.96, 41.75, 41.04) mm, rotated rx 180 ry 0 rz 180 deg; joints [-18.313, 15.866, 50.103, 39.103, 29.88, -35.173]
  Call Extruder(199.20245)
  MoveL 1937 to (238.13, 41.99, 41.04) mm, rotated rx -180 ry 0 rz 180 deg; joints [-18.333, 15.917, 50.038, 39.119, 29.903, -35.182]
  MoveL 1938 to (238.13, 41.99, 41.04) mm, rotated rx -180 ry 0 rz 180 deg; joints [-18.333, 15.917, 50.038, 39.119, 29.903, -35.182]
  Call Extruder(199.41057)
  MoveL 1939 to (238.31, 42.3, 41.04) mm, rotated rx -180 ry 0 rz 180 deg; joints [-18.36, 15.971, 49.967, 39.144, 29.931, -35.199]
  MoveL 1940 to (238.31, 42.3, 41.04) mm, rotated rx -180 ry 0 rz 180 deg; joints [-18.36, 15.971, 49.967, 39.144, 29.931, -35.199]
  Call Extruder(199.61791)
  MoveL 1941 to (238.49, 42.6, 41.04) mm, rotated rx -180 ry 0 rz 180 deg; joints [-18.386, 16.025, 49.896, 39.169, 29.959, -35.215]
  MoveL 1942 to (238.49, 42.6, 41.04) mm, rotated rx -180 ry 0 rz 180 deg; joints [-18.386, 16.025, 49.896, 39.169, 29.959, -35.215]
  Call Extruder(199.82447)
  MoveL 1943 to (238.66, 42.91, 41.04) mm, rotated rx -180 ry 0 rz 180 deg; joints [-18.412, 16.08, 49.825, 39.194, 29.987, -35.232]
  MoveL 1944 to (238.66, 42.91, 41.04) mm, rotated rx -180 ry 0 rz 180 deg; joints [-18.412, 16.08, 49.825, 39.194, 29.987, -35.232]
  Call Extruder(200.03025)
  MoveL 1945 to (238.84, 43.21, 41.03) mm, rotated rx -180 ry 0 rz 180 deg; joints [-18.438, 16.135, 49.754, 39.218, 30.015, -35.248]
  MoveL 1946 to (238.84, 43.21, 41.03) mm, rotated rx -180 ry 0 rz 180 deg; joints [-18.438, 16.135, 49.754, 39.218, 30.015, -35.248]
  Call Extruder(200.18856)
  MoveL 1947 to (238.94, 43.46, 41.04) mm, rotated rx 180 ry 0 rz 180 deg; joints [-18.461, 16.172, 49.705, 39.243, 30.037, -35.266]
  MoveL 1948 to (238.94, 43.46, 41.04) mm, rotated rx 180 ry 0 rz 180 deg; joints [-18.461, 16.172, 49.705, 39.243, 30.037, -35.266]
  Call Extruder(200.34626)
  MoveL 1949 to (239.05, 43.71, 41.04) mm, rotated rx 180 ry 0 rz 180 deg; joints [-18.484, 16.21, 49.655, 39.268, 30.059, -35.283]
  MoveL 1950 to (239.05, 43.71, 41.04) mm, rotated rx 180 ry 0 rz 180 deg; joints [-18.484, 16.21, 49.655, 39.268, 30.059, -35.283]
  Call Extruder(200.51634)
  MoveL 1951 to (239.17, 43.98, 41.03) mm, rotated rx 180 ry 0 rz 180 deg; joints [-18.509, 16.25, 49.603, 39.294, 30.083, -35.302]
  MoveL 1952 to (239.17, 43.98, 41.03) mm, rotated rx 180 ry 0 rz 180 deg; joints [-18.509, 16.25, 49.603, 39.294, 30.083, -35.302]
  Call Extruder(200.69866)
  MoveL 1953 to (239.29, 44.27, 41.04) mm, rotated rx 180 ry 0 rz -180 deg; joints [-18.535, 16.294, 49.546, 39.323, 30.109, -35.323]
  MoveL 1954 to (239.29, 44.27, 41.04) mm, rotated rx 180 ry 0 rz -180 deg; joints [-18.535, 16.294, 49.546, 39.323, 30.109, -35.323]
  Call Extruder(200.88022)
  MoveL 1955 to (239.41, 44.56, 41.04) mm, rotated rx 180 ry 0 rz 180 deg; joints [-18.562, 16.337, 49.489, 39.352, 30.135, -35.344]
  MoveL 1956 to (239.41, 44.56, 41.04) mm, rotated rx 180 ry 0 rz 180 deg; joints [-18.562, 16.337, 49.489, 39.352, 30.135, -35.344]
  Call Extruder(200.93707)
  MoveL 1957 to (239.44, 44.66, 41.04) mm, rotated rx -180 ry 0 rz 180 deg; joints [-18.571, 16.349, 49.473, 39.363, 30.143, -35.352]
  MoveL 1958 to (239.44, 44.66, 41.04) mm, rotated rx -180 ry 0 rz 180 deg; joints [-18.571, 16.349, 49.473, 39.363, 30.143, -35.352]
  Call Extruder(201.05031)
  MoveL 1959 to (239.5, 44.85, 41.04) mm, rotated rx -180 ry 0 rz 180 deg; joints [-18.589, 16.374, 49.44, 39.383, 30.159, -35.367]
  MoveL 1960 to (239.5, 44.85, 41.04) mm, rotated rx -180 ry 0 rz 180 deg; joints [-18.589, 16.374, 49.44, 39.383, 30.159, -35.367]
  Call Extruder(201.16311)
  MoveL 1961 to (239.56, 45.03, 41.04) mm, rotated rx 180 ry 0 rz 180 deg; joints [-18.607, 16.399, 49.408, 39.404, 30.175, -35.382]
  MoveL 1962 to (239.56, 45.03, 41.04) mm, rotated rx 180 ry 0 rz 180 deg; joints [-18.607, 16.399, 49.408, 39.404, 30.175, -35.382]
  Call Extruder(201.27546)
  MoveL 1963 to (239.62, 45.22, 41.04) mm, rotated rx 180 ry 0 rz 180 deg; joints [-18.625, 16.424, 49.376, 39.425, 30.192, -35.398]
  MoveL 1964 to (239.62, 45.22, 41.04) mm, rotated rx 180 ry 0 rz 180 deg; joints [-18.625, 16.424, 49.376, 39.425, 30.192, -35.398]
  Call Extruder(201.38737)
  MoveL 1965 to (239.68, 45.41, 41.04) mm, rotated rx 180 ry 0 rz 180 deg; joints [-18.642, 16.448, 49.343, 39.445, 30.208, -35.413]
  MoveL 1966 to (239.68, 45.41, 41.04) mm, rotated rx 180 ry 0 rz 180 deg; joints [-18.642, 16.448, 49.343, 39.445, 30.208, -35.413]
  Call Extruder(201.50878)
  MoveL 1967 to (239.75, 45.62, 41.04) mm, rotated rx -180 ry 0 rz 180 deg; joints [-18.662, 16.475, 49.308, 39.468, 30.226, -35.43]
  MoveL 1968 to (239.75, 45.62, 41.04) mm, rotated rx -180 ry 0 rz 180 deg; joints [-18.662, 16.475, 49.308, 39.468, 30.226, -35.43]
  Call Extruder(201.63957)
  MoveL 1969 to (239.82, 45.84, 41.04) mm, rotated rx 180 ry 0 rz 180 deg; joints [-18.683, 16.504, 49.271, 39.492, 30.245, -35.448]
  MoveL 1970 to (239.82, 45.84, 41.04) mm, rotated rx 180 ry 0 rz 180 deg; joints [-18.683, 16.504, 49.271, 39.492, 30.245, -35.448]
  Call Extruder(201.76979)
  MoveL 1971 to (239.88, 46.06, 41.04) mm, rotated rx 180 ry 0 rz 180 deg; joints [-18.705, 16.532, 49.233, 39.517, 30.264, -35.467]
  MoveL 1972 to (239.88, 46.06, 41.04) mm, rotated rx 180 ry 0 rz 180 deg; joints [-18.705, 16.532, 49.233, 39.517, 30.264, -35.467]
  Call Extruder(201.89946)
  MoveL 1973 to (239.95, 46.29, 41.04) mm, rotated rx 180 ry 0 rz 180 deg; joints [-18.726, 16.561, 49.196, 39.542, 30.283, -35.485]
  MoveL 1974 to (239.95, 46.29, 41.04) mm, rotated rx 180 ry 0 rz 180 deg; joints [-18.726, 16.561, 49.196, 39.542, 30.283, -35.485]
  Call Extruder(202.02855)
  MoveL 1975 to (240.02, 46.51, 41.04) mm, rotated rx 180 ry 0 rz 180 deg; joints [-18.747, 16.589, 49.158, 39.567, 30.303, -35.504]
  MoveL 1976 to (240.02, 46.51, 41.04) mm, rotated rx 180 ry 0 rz 180 deg; joints [-18.747, 16.589, 49.158, 39.567, 30.303, -35.504]
  Call Extruder(202.14360)
  MoveL 1977 to (240.06, 46.72, 41.04) mm, rotated rx 180 ry 0 rz 180 deg; joints [-18.767, 16.612, 49.128, 39.591, 30.32, -35.523]
  MoveL 1978 to (240.06, 46.72, 41.04) mm, rotated rx 180 ry 0 rz 180 deg; joints [-18.767, 16.612, 49.128, 39.591, 30.32, -35.523]
  Call Extruder(202.25820)
  MoveL 1979 to (240.11, 46.92, 41.03) mm, rotated rx 180 ry 0 rz 180 deg; joints [-18.787, 16.635, 49.098, 39.615, 30.337, -35.541]
  MoveL 1980 to (240.11, 46.92, 41.03) mm, rotated rx 180 ry 0 rz 180 deg; joints [-18.787, 16.635, 49.098, 39.615, 30.337, -35.541]
  Call Extruder(202.37235)
  MoveL 1981 to (240.15, 47.12, 41.03) mm, rotated rx 180 ry 0 rz 180 deg; joints [-18.807, 16.658, 49.069, 39.64, 30.354, -35.56]
  MoveL 1982 to (240.15, 47.12, 41.03) mm, rotated rx 180 ry 0 rz 180 deg; joints [-18.807, 16.658, 49.069, 39.64, 30.354, -35.56]
  Call Extruder(202.48605)
  MoveL 1983 to (240.2, 47.33, 41.04) mm, rotated rx -180 ry 0 rz 180 deg; joints [-18.827, 16.681, 49.038, 39.664, 30.371, -35.579]
  MoveL 1984 to (240.2, 47.33, 41.04) mm, rotated rx -180 ry 0 rz 180 deg; joints [-18.827, 16.681, 49.038, 39.664, 30.371, -35.579]
  Call Extruder(202.61146)
  MoveL 1985 to (240.24, 47.56, 41.04) mm, rotated rx -180 ry 0 rz 180 deg; joints [-18.85, 16.706, 49.006, 39.692, 30.39, -35.6]
  MoveL 1986 to (240.24, 47.56, 41.04) mm, rotated rx -180 ry 0 rz 180 deg; joints [-18.85, 16.706, 49.006, 39.692, 30.39, -35.6]
  Call Extruder(202.74844)
  MoveL 1987 to (240.29, 47.8, 41.04) mm, rotated rx -180 ry 0 rz 180 deg; joints [-18.874, 16.733, 48.97, 39.722, 30.411, -35.623]
  MoveL 1988 to (240.29, 47.8, 41.04) mm, rotated rx -180 ry 0 rz 180 deg; joints [-18.874, 16.733, 48.97, 39.722, 30.411, -35.623]
  Call Extruder(202.88480)
  MoveL 1989 to (240.34, 48.05, 41.04) mm, rotated rx 180 ry 0 rz 180 deg; joints [-18.899, 16.759, 48.935, 39.752, 30.432, -35.647]
  MoveL 1990 to (240.34, 48.05, 41.04) mm, rotated rx 180 ry 0 rz 180 deg; joints [-18.899, 16.759, 48.935, 39.752, 30.432, -35.647]
  Call Extruder(203.02056)
  MoveL 1991 to (240.39, 48.3, 41.04) mm, rotated rx 180 ry 0 rz 180 deg; joints [-18.923, 16.787, 48.899, 39.782, 30.453, -35.67]
  MoveL 1992 to (240.39, 48.3, 41.04) mm, rotated rx 180 ry 0 rz 180 deg; joints [-18.923, 16.787, 48.899, 39.782, 30.453, -35.67]
  Call Extruder(203.15571)
  MoveL 1993 to (240.44, 48.55, 41.04) mm, rotated rx 180 ry 0 rz 180 deg; joints [-18.948, 16.814, 48.863, 39.812, 30.474, -35.693]
  MoveL 1994 to (240.44, 48.55, 41.04) mm, rotated rx 180 ry 0 rz 180 deg; joints [-18.948, 16.814, 48.863, 39.812, 30.474, -35.693]
  Call Extruder(203.29025)
  MoveL 1995 to (240.49, 48.8, 41.04) mm, rotated rx -180 ry 0 rz 180 deg; joints [-18.973, 16.841, 48.828, 39.842, 30.495, -35.716]
  MoveL 1996 to (240.49, 48.8, 41.04) mm, rotated rx -180 ry 0 rz 180 deg; joints [-18.973, 16.841, 48.828, 39.842, 30.495, -35.716]
  Call Extruder(203.42417)
  MoveL 1997 to (240.54, 49.05, 41.04) mm, rotated rx -180 ry 0 rz 180 deg; joints [-18.997, 16.868, 48.792, 39.872, 30.516, -35.739]
  MoveL 1998 to (240.54, 49.05, 41.04) mm, rotated rx -180 ry 0 rz 180 deg; joints [-18.997, 16.868, 48.792, 39.872, 30.516, -35.739]
  Call Extruder(203.57204)
  MoveL 1999 to (240.59, 49.33, 41.04) mm, rotated rx -180 ry 0 rz 180 deg; joints [-19.025, 16.897, 48.754, 39.906, 30.539, -35.765]
  MoveL 2000 to (240.59, 49.33, 41.04) mm, rotated rx -180 ry 0 rz 180 deg; joints [-19.025, 16.897, 48.754, 39.906, 30.539, -35.765]
  Call Extruder(203.73378)
  MoveL 2001 to (240.64, 49.63, 41.03) mm, rotated rx -180 ry 0 rz 180 deg; joints [-19.055, 16.928, 48.713, 39.943, 30.564, -35.794]
  MoveL 2002 to (240.64, 49.63, 41.03) mm, rotated rx -180 ry 0 rz 180 deg; joints [-19.055, 16.928, 48.713, 39.943, 30.564, -35.794]
  Call Extruder(203.89480)
  MoveL 2003 to (240.69, 49.94, 41.03) mm, rotated rx -180 ry 0 rz 180 deg; joints [-19.086, 16.959, 48.672, 39.981, 30.59, -35.824]
  MoveL 2004 to (240.69, 49.94, 41.03) mm, rotated rx -180 ry 0 rz 180 deg; joints [-19.086, 16.959, 48.672, 39.981, 30.59, -35.824]
  Call Extruder(204.05509)
  MoveL 2005 to (240.74, 50.24, 41.03) mm, rotated rx 180 ry 0 rz 180 deg; joints [-19.116, 16.99, 48.631, 40.019, 30.615, -35.853]
  MoveL 2006 to (240.74, 50.24, 41.03) mm, rotated rx 180 ry 0 rz 180 deg; joints [-19.116, 16.99, 48.631, 40.019, 30.615, -35.853]
  Call Extruder(204.21465)
  MoveL 2007 to (240.78, 50.55, 41.04) mm, rotated rx -180 ry 0 rz 180 deg; joints [-19.146, 17.021, 48.59, 40.057, 30.641, -35.882]
  MoveL 2008 to (240.78, 50.55, 41.04) mm, rotated rx -180 ry 0 rz 180 deg; joints [-19.146, 17.021, 48.59, 40.057, 30.641, -35.882]
  Call Extruder(204.37349)
  MoveL 2009 to (240.83, 50.86, 41.04) mm, rotated rx -180 ry 0 rz -180 deg; joints [-19.177, 17.052, 48.548, 40.094, 30.666, -35.911]
  MoveL 2010 to (240.83, 50.86, 41.04) mm, rotated rx -180 ry 0 rz -180 deg; joints [-19.177, 17.052, 48.548, 40.094, 30.666, -35.911]
  Call Extruder(204.55216)
  MoveL 2011 to (240.88, 51.2, 41.03) mm, rotated rx -180 ry 0 rz 180 deg; joints [-19.212, 17.086, 48.504, 40.137, 30.695, -35.944]
  MoveL 2012 to (240.88, 51.2, 41.03) mm, rotated rx -180 ry 0 rz 180 deg; joints [-19.212, 17.086, 48.504, 40.137, 30.695, -35.944]
  Call Extruder(204.75060)
  MoveL 2013 to (240.92, 51.59, 41.04) mm, rotated rx 180 ry 0 rz 180 deg; joints [-19.251, 17.123, 48.455, 40.186, 30.727, -35.983]
  MoveL 2014 to (240.92, 51.59, 41.04) mm, rotated rx 180 ry 0 rz 180 deg; joints [-19.251, 17.123, 48.455, 40.186, 30.727, -35.983]
  Call Extruder(204.94818)
  MoveL 2015 to (240.97, 51.98, 41.04) mm, rotated rx -180 ry 0 rz 180 deg; joints [-19.29, 17.159, 48.407, 40.235, 30.759, -36.021]
  MoveL 2016 to (240.97, 51.98, 41.04) mm, rotated rx -180 ry 0 rz 180 deg; joints [-19.29, 17.159, 48.407, 40.235, 30.759, -36.021]
  Call Extruder(205.14488)
  MoveL 2017 to (241.02, 52.37, 41.04) mm, rotated rx 180 ry 0 rz 180 deg; joints [-19.329, 17.196, 48.358, 40.284, 30.791, -36.059]
  MoveL 2018 to (241.02, 52.37, 41.04) mm, rotated rx 180 ry 0 rz 180 deg; joints [-19.329, 17.196, 48.358, 40.284, 30.791, -36.059]
  Call Extruder(205.34072)
  MoveL 2019 to (241.06, 52.75, 41.04) mm, rotated rx 180 ry 0 rz 180 deg; joints [-19.368, 17.232, 48.309, 40.333, 30.823, -36.096]
  MoveL 2020 to (241.06, 52.75, 41.04) mm, rotated rx 180 ry 0 rz 180 deg; joints [-19.368, 17.232, 48.309, 40.333, 30.823, -36.096]
  Call Extruder(205.63616)
  MoveL 2021 to (241.11, 53.34, 41.03) mm, rotated rx 180 ry 0 rz 180 deg; joints [-19.428, 17.284, 48.241, 40.409, 30.872, -36.157]
  MoveL 2022 to (241.11, 53.34, 41.03) mm, rotated rx 180 ry 0 rz 180 deg; joints [-19.428, 17.284, 48.241, 40.409, 30.872, -36.157]
  Call Extruder(205.93027)
  MoveL 2023 to (241.15, 53.93, 41.04) mm, rotated rx -180 ry 0 rz 180 deg; joints [-19.488, 17.336, 48.173, 40.485, 30.92, -36.216]
  MoveL 2024 to (241.15, 53.93, 41.04) mm, rotated rx -180 ry 0 rz 180 deg; joints [-19.488, 17.336, 48.173, 40.485, 30.92, -36.216]
  Call Extruder(206.22304)
  MoveL 2025 to (241.2, 54.52, 41.04) mm, rotated rx 180 ry 0 rz 180 deg; joints [-19.548, 17.387, 48.104, 40.561, 30.969, -36.276]
  MoveL 2026 to (241.2, 54.52, 41.04) mm, rotated rx 180 ry 0 rz 180 deg; joints [-19.548, 17.387, 48.104, 40.561, 30.969, -36.276]
  Call Extruder(206.79649)
  MoveL 2027 to (241.25, 55.68, 41.04) mm, rotated rx 180 ry 0 rz -180 deg; joints [-19.668, 17.481, 47.979, 40.715, 31.063, -36.397]
  MoveL 2028 to (241.25, 55.68, 41.04) mm, rotated rx 180 ry 0 rz -180 deg; joints [-19.668, 17.481, 47.979, 40.715, 31.063, -36.397]
  Call Extruder(207.51032)
